FUNCTION_BLOCK "Sq_5.1"   // FB1511, GRAPH_PLUS
{ S7_Optimized_Access := 'TRUE' }
VERSION : 0.1
   VAR_INPUT
      OFF_SQ : Bool := false;   // Kette ausschalten
      INIT_SQ : Bool := false;   // Kette in Initialzustand versetzen
      ACK_EF : Bool := false;   // Alle Fehler und Störungen quittieren
      S_PREV : Bool := false;   // Vorherigen Schritt am Parameter S_NO ausgeben
      S_NEXT : Bool := false;   // Nächsten Schritt am Parameter S_NO anzeigen
      SW_AUTO : Bool := false;   // Automatischer Betrieb
      SW_TAP : Bool := false;   // Halbautomatisch/Weiterschalten mit Transition
      SW_TOP : Bool := false;   // Halbautomatisch/Ignoriere Transition
      SW_MAN : Bool := false;   // Handbetrieb
      S_SEL : Int := 0;   // Schritt auswählen, der an S_NO ausgegeben werden soll
      S_ON : Bool := false;   // Schritt aktivieren, der an Parameter S_NO anliegt
      S_OFF : Bool := false;   // Schritt deaktivieren, der an Parameter S_NO anliegt
      T_PUSH : Bool := false;   // Schaltfreigabe für Transition im halbautomatischen Betrieb
      itMaxRuntime : Time := t#10s;   // Maximale Laufzeit für diesen Prozess
   END_VAR
   VAR_OUTPUT
      S_NO : Int := 0;   // Schrittnummer
      S_MORE : Bool := false;   // Weitere Schritte sind vorhanden und können in S_NO angezeigt werden.
      S_ACTIVE : Bool := false;   // Schritt, der an Parameter S_NO angezeigt wird, ist aktiv
      ERR_FLT : Bool := false;   // Sammelfehler Interlock oder Supervision
      AUTO_ON : Bool := false;   // Automatischer Betrieb eingeschaltet
      TAP_ON : Bool := false;   // Halbautomatischer Betrieb/Schritt mit Transition eingeschaltet
      TOP_ON : Bool := false;   // Halbautomatischer Betrieb/Ignoriere Transition eingeschaltet
      MAN_ON : Bool := false;   // Handbetrieb eingeschaltet
      qxIsActive : Bool;   // Schrittkette läuft
      qxIsInHome : Bool;   // steht in Grundstellung
      qxConveyorIsEmpty : Bool;   // Linearförderer wurde geleert
      qxLackOfParts : Bool;   // Teilemangel
   END_VAR
   VAR_IN_OUT
      signals : "typeStationSignals";   // Stationssteuersignale
      sq : "typeStepSequence";   // Schrittkettensteuersignale
   END_VAR
   VAR
      sstReleaseCycle : Struct
         ErrorAck : Bool;
         No_LastCycle : Int;
         T : Time;   // Aktive Zeit des ReleaseCycle
         Tck : Time;
         TckPrev : Time;
      END_STRUCT;
      susiGripperState : USInt;
      sinstTofConveyorOn : TOF_TIME;
      sinstTonConveyorIsEmpty : TON_TIME;
      sinstTonPartInSep : TON_TIME;
      sinstTonLackOfParts : TON_TIME;
      sinstTonNoPartInSep : TON_TIME;
      sxConveyorOn : Bool;
      sxWaitForPart : Bool;
      HMI_INFO : Array[0..8] of UInt;
      IF_PAR : G7_IfParPlus_V6;
      RT_DATA : G7_RTDataPlus_V6;   // Interner Datenbereich
      Automatikablauf : G7_TransitionPlus_V6;   // Transitionsstruktur
      Freigabe : G7_TransitionPlus_V6;   // Transitionsstruktur
      GreiferLeer : G7_TransitionPlus_V6;   // Transitionsstruktur
      Fertig : G7_TransitionPlus_V6;   // Transitionsstruktur
      Grundstellungsfahrt : G7_TransitionPlus_V6;   // Transitionsstruktur
      GST_Aktiv : G7_TransitionPlus_V6;   // Transitionsstruktur
      GST_Beendet : G7_TransitionPlus_V6;   // Transitionsstruktur
      Beendet : G7_TransitionPlus_V6;   // Transitionsstruktur
      DoneToIndexer : G7_TransitionPlus_V6;   // Transitionsstruktur / Transition structure
      JogT1 : G7_TransitionPlus_V6;   // Transitionsstruktur / Transition structure
      JogT2 : G7_TransitionPlus_V6;   // Transitionsstruktur / Transition structure
      GS_CapsSourceStopperInHome : G7_TransitionPlus_V6;   // Transitionsstruktur / Transition structure
      GS_NotEmptying : G7_TransitionPlus_V6;   // Transitionsstruktur / Transition structure
      GS_Emptying : G7_TransitionPlus_V6;   // Transitionsstruktur / Transition structure
      GS_CapsSourceStopperInWork : G7_TransitionPlus_V6;   // Transitionsstruktur / Transition structure
      GS_AxisRInHome : G7_TransitionPlus_V6;   // Transitionsstruktur / Transition structure
      GS_AxisZ1InHome : G7_TransitionPlus_V6;   // Transitionsstruktur / Transition structure
      GS_AxisZ2InHome : G7_TransitionPlus_V6;   // Transitionsstruktur / Transition structure
      GS_AxisXInHome : G7_TransitionPlus_V6;   // Transitionsstruktur / Transition structure
      GS_GreiferUnbeladen : G7_TransitionPlus_V6;   // Transitionsstruktur / Transition structure
      GS_GreiferBeladen : G7_TransitionPlus_V6;   // Transitionsstruktur / Transition structure
      GS_GreiferUnbekannt : G7_TransitionPlus_V6;   // Transitionsstruktur / Transition structure
      GS_GripperInHome : G7_TransitionPlus_V6;   // Transitionsstruktur / Transition structure
      GS_GripperInWork : G7_TransitionPlus_V6;   // Transitionsstruktur / Transition structure
      GS_CapsSourceStopperInWork_1 : G7_TransitionPlus_V6;   // Transitionsstruktur / Transition structure
      GS_GripperInHome_1 : G7_TransitionPlus_V6;   // Transitionsstruktur / Transition structure
      CapsSourceStopperInHome_1 : G7_TransitionPlus_V6;   // Transitionsstruktur / Transition structure
      GS_GripperStatusIsEmpty : G7_TransitionPlus_V6;   // Transitionsstruktur / Transition structure
      NotEmptying : G7_TransitionPlus_V6;   // Transitionsstruktur / Transition structure
      Emptying : G7_TransitionPlus_V6;   // Transitionsstruktur / Transition structure
      CapsSourceStopperInWork_2 : G7_TransitionPlus_V6;   // Transitionsstruktur / Transition structure
      GripperInHome_2 : G7_TransitionPlus_V6;   // Transitionsstruktur / Transition structure
      GripperIsEmpty : G7_TransitionPlus_V6;   // Transitionsstruktur / Transition structure
      ConveyorIsEmpty : G7_TransitionPlus_V6;   // Transitionsstruktur / Transition structure
      SepEmpty : G7_TransitionPlus_V6;   // Transitionsstruktur / Transition structure
      SepNotEmpty : G7_TransitionPlus_V6;   // Transitionsstruktur / Transition structure
      CapsSourceStopperInHome : G7_TransitionPlus_V6;   // Transitionsstruktur / Transition structure
      AxisZ2InWork : G7_TransitionPlus_V6;   // Transitionsstruktur / Transition structure
      GripperInWork : G7_TransitionPlus_V6;   // Transitionsstruktur / Transition structure
      GripperIsLoaded : G7_TransitionPlus_V6;   // Transitionsstruktur / Transition structure
      AxisZ2InHome : G7_TransitionPlus_V6;   // Transitionsstruktur / Transition structure
      JogT3 : G7_TransitionPlus_V6;   // Transitionsstruktur / Transition structure
      JogT4 : G7_TransitionPlus_V6;   // Transitionsstruktur / Transition structure
      JogT5 : G7_TransitionPlus_V6;   // Transitionsstruktur / Transition structure
      SeparatorIsEmpty : G7_TransitionPlus_V6;   // Transitionsstruktur / Transition structure
      ConvEmptyIsSet : G7_TransitionPlus_V6;   // Transitionsstruktur / Transition structure
      JogT6 : G7_TransitionPlus_V6;   // Transitionsstruktur / Transition structure
      GripperIsLoaded_1 : G7_TransitionPlus_V6;   // Transitionsstruktur / Transition structure
      GripperIsEmpty_1 : G7_TransitionPlus_V6;   // Transitionsstruktur / Transition structure
      CapsSourceStopperInHome_2 : G7_TransitionPlus_V6;   // Transitionsstruktur / Transition structure
      GripperInWork_1 : G7_TransitionPlus_V6;   // Transitionsstruktur / Transition structure
      GripperIsLoaded_2 : G7_TransitionPlus_V6;   // Transitionsstruktur / Transition structure
      PartInSeparator_2 : G7_TransitionPlus_V6;   // Transitionsstruktur / Transition structure
      AxisZ2InWork_2 : G7_TransitionPlus_V6;   // Transitionsstruktur / Transition structure
      AxisZ2InHome_1 : G7_TransitionPlus_V6;   // Transitionsstruktur / Transition structure
      SeparatorIsEmpty_1 : G7_TransitionPlus_V6;   // Transitionsstruktur / Transition structure
      JogT7 : G7_TransitionPlus_V6;   // Transitionsstruktur / Transition structure
      JogT8 : G7_TransitionPlus_V6;   // Transitionsstruktur / Transition structure
      JogT9 : G7_TransitionPlus_V6;   // Transitionsstruktur / Transition structure
      AxisXInWork : G7_TransitionPlus_V6;   // Transitionsstruktur / Transition structure
      AxisRInWork : G7_TransitionPlus_V6;   // Transitionsstruktur / Transition structure
      AxisZ1InWork : G7_TransitionPlus_V6;   // Transitionsstruktur / Transition structure
      GripperInHome_3 : G7_TransitionPlus_V6;   // Transitionsstruktur / Transition structure
      GripperIsEmpty_2 : G7_TransitionPlus_V6;   // Transitionsstruktur / Transition structure
      AxisZ1InHome : G7_TransitionPlus_V6;   // Transitionsstruktur / Transition structure
      GS_AxisRInHome_1 : G7_TransitionPlus_V6;   // Transitionsstruktur / Transition structure
      AxisXInHome : G7_TransitionPlus_V6;   // Transitionsstruktur / Transition structure
      JogT10 : G7_TransitionPlus_V6;   // Transitionsstruktur / Transition structure
      JogT11 : G7_TransitionPlus_V6;   // Transitionsstruktur / Transition structure
      JogT12 : G7_TransitionPlus_V6;   // Transitionsstruktur / Transition structure
      JogT13 : G7_TransitionPlus_V6;   // Transitionsstruktur / Transition structure
      JogT14 : G7_TransitionPlus_V6;   // Transitionsstruktur / Transition structure
      JogT15 : G7_TransitionPlus_V6;   // Transitionsstruktur / Transition structure
      Initialschritt : G7_StepPlus_V6;   // Schrittstruktur
      Grundstellung : G7_StepPlus_V6;   // Schrittstruktur
      SK_läuft : G7_StepPlus_V6;   // Schrittstruktur
      Fertigmeldung : G7_StepPlus_V6;   // Schrittstruktur
      "Start Grundstellungsfahrt" : G7_StepPlus_V6;   // Schrittstruktur
      "Fertig Grundstellungsfahrt" : G7_StepPlus_V6;   // Schrittstruktur
      Ende : G7_StepPlus_V6;   // Schrittstruktur
      ResetRelease : G7_StepPlus_V6;   // Schrittstruktur / Step structure
      JogS1 : G7_StepPlus_V6;   // Schrittstruktur / Step structure
      JogS2 : G7_StepPlus_V6;   // Schrittstruktur / Step structure
      GS_CapsSourceStopperHomePos : G7_StepPlus_V6;   // Schrittstruktur / Step structure
      "GS_Emptying?" : G7_StepPlus_V6;   // Schrittstruktur / Step structure
      GS_CapsSourceStopperWorkPos : G7_StepPlus_V6;   // Schrittstruktur / Step structure
      GS_AxisRHomePos : G7_StepPlus_V6;   // Schrittstruktur / Step structure
      GS_AxisZ1HomePos : G7_StepPlus_V6;   // Schrittstruktur / Step structure
      GS_AxisZ2HomePos : G7_StepPlus_V6;   // Schrittstruktur / Step structure
      GS_AxisXHomePos : G7_StepPlus_V6;   // Schrittstruktur / Step structure
      GS_GripperState : G7_StepPlus_V6;   // Schrittstruktur / Step structure
      GS_GripperHomePos : G7_StepPlus_V6;   // Schrittstruktur / Step structure
      GS_GripperWorkPos : G7_StepPlus_V6;   // Schrittstruktur / Step structure
      GS_CapsSourceStopperWorkPos_1 : G7_StepPlus_V6;   // Schrittstruktur / Step structure
      GS_GripperHomePos_1 : G7_StepPlus_V6;   // Schrittstruktur / Step structure
      GS_CapsSourceStopperHomePos_1 : G7_StepPlus_V6;   // Schrittstruktur / Step structure
      GS_GripperStatusEmpty : G7_StepPlus_V6;   // Schrittstruktur / Step structure
      "Emptying?" : G7_StepPlus_V6;   // Schrittstruktur / Step structure
      CapsSourceStopperWorkPos : G7_StepPlus_V6;   // Schrittstruktur / Step structure
      GripperHomePos : G7_StepPlus_V6;   // Schrittstruktur / Step structure
      GripperEmpty : G7_StepPlus_V6;   // Schrittstruktur / Step structure
      EmptyingConveyor : G7_StepPlus_V6;   // Schrittstruktur / Step structure
      SeparatorEmpty : G7_StepPlus_V6;   // Schrittstruktur / Step structure
      CapsSourceStopperHomePos : G7_StepPlus_V6;   // Schrittstruktur / Step structure
      AxisZ2WorkPos : G7_StepPlus_V6;   // Schrittstruktur / Step structure
      GripperWorkPos : G7_StepPlus_V6;   // Schrittstruktur / Step structure
      GripperLoaded : G7_StepPlus_V6;   // Schrittstruktur / Step structure
      AxisZ2HomePos : G7_StepPlus_V6;   // Schrittstruktur / Step structure
      JogS3 : G7_StepPlus_V6;   // Schrittstruktur / Step structure
      JogS4 : G7_StepPlus_V6;   // Schrittstruktur / Step structure
      JogS5 : G7_StepPlus_V6;   // Schrittstruktur / Step structure
      CheckSepEmpty : G7_StepPlus_V6;   // Schrittstruktur / Step structure
      SetConvEmpty : G7_StepPlus_V6;   // Schrittstruktur / Step structure
      JogS6 : G7_StepPlus_V6;   // Schrittstruktur / Step structure
      GripperState : G7_StepPlus_V6;   // Schrittstruktur / Step structure
      CapsSourceStopperHomePos_1 : G7_StepPlus_V6;   // Schrittstruktur / Step structure
      GripperWorkPos_1 : G7_StepPlus_V6;   // Schrittstruktur / Step structure
      GripperLoaded_1 : G7_StepPlus_V6;   // Schrittstruktur / Step structure
      SeparatorBusy_1 : G7_StepPlus_V6;   // Schrittstruktur / Step structure
      AxisZ2WorkPos_2 : G7_StepPlus_V6;   // Schrittstruktur / Step structure
      AxisZ2HomePos_1 : G7_StepPlus_V6;   // Schrittstruktur / Step structure
      CheckSepEmpty_1 : G7_StepPlus_V6;   // Schrittstruktur / Step structure
      JogS7 : G7_StepPlus_V6;   // Schrittstruktur / Step structure
      JogS8 : G7_StepPlus_V6;   // Schrittstruktur / Step structure
      JogS9 : G7_StepPlus_V6;   // Schrittstruktur / Step structure
      AxisXWorkPos : G7_StepPlus_V6;   // Schrittstruktur / Step structure
      AxisRWorkPos : G7_StepPlus_V6;   // Schrittstruktur / Step structure
      AxisZ1WorkPos : G7_StepPlus_V6;   // Schrittstruktur / Step structure
      GripperHomePos_1 : G7_StepPlus_V6;   // Schrittstruktur / Step structure
      GripperEmpty_1 : G7_StepPlus_V6;   // Schrittstruktur / Step structure
      AxisZ1HomePos : G7_StepPlus_V6;   // Schrittstruktur / Step structure
      GS_AxisRHomePos_1 : G7_StepPlus_V6;   // Schrittstruktur / Step structure
      AxisXHomePos : G7_StepPlus_V6;   // Schrittstruktur / Step structure
      JogS10 : G7_StepPlus_V6;   // Schrittstruktur / Step structure
      JogS11 : G7_StepPlus_V6;   // Schrittstruktur / Step structure
      JogS12 : G7_StepPlus_V6;   // Schrittstruktur / Step structure
      JogS13 : G7_StepPlus_V6;   // Schrittstruktur / Step structure
      JogS14 : G7_StepPlus_V6;   // Schrittstruktur / Step structure
      JogS15 : G7_StepPlus_V6;   // Schrittstruktur / Step structure
      SINI : Array[0..1] of USInt;
      LSTT : Array[0..72] of USInt;
      ATAJ : Array[0..72] of USInt;
      ATAB : Array[0..72] of USInt;
      PSTT : Array[0..72] of USInt;
      NSTT : Array[0..72] of USInt;
      ASSJ : Array[0..65] of USInt;
      ASSB : Array[0..65] of USInt;
      PTTS : Array[0..65] of USInt;
      NTTS : Array[0..65] of USInt;
      SW_SQTS : Array[0..65] of USInt;
      SWITCH : Array[0..40] of USInt;
      TVX : Array[0..14] of USInt;
      TTX : Array[0..14] of USInt;
      TSX : Array[0..1] of USInt;
      S00X : Array[0..1] of USInt;
      SOFFX : Array[0..1] of USInt;
      SONX : Array[0..1] of USInt;
      SAX : Array[0..1] of USInt;
      SERRX : Array[0..66] of USInt;
      SMX : Array[0..66] of USInt;
      S0X : Array[0..66] of USInt;
      S1X : Array[0..66] of USInt;
      IL_ALARM_INST : Diag_Alarm;
      SUP_ALARM_INST : Diag_Alarm;
      STEP_TIME_ALARM_INST : Diag_Alarm;
      IEC_TIMER_INST : IEC_TIMER;
      TRANSACTION_FLAG : Bool := false;
   END_VAR
   VAR_TEMP
      txStartCondition : Bool;
      tdTckDiff : DInt;
   END_VAR
   VAR CONSTANT
      GRIPPER_UNKNOWN : USInt := 0;   // Greiferstatus "unbekannt"
      GRIPPER_EMPTY : USInt := 1;   // Greiferstatus "leer"
      GRIPPER_LOADED : USInt := 2;   // Greiferstatus "beladen"
   END_VAR
   VAR_TEMP   // added for the SCL form of the ladder/FBD networks
      _w1 : Bool;
      _w2 : Bool;
   END_VAR
   // SINI[0] := 2;
   // LSTT[0] := 255;
   // LSTT[1] := 255;
   // LSTT[2] := 255;
   // LSTT[3] := 255;
   // LSTT[4] := 255;
   // LSTT[5] := 255;
   // LSTT[6] := 255;
   // LSTT[7] := 1;
   // ATAJ[1] := 1;
   // ATAJ[2] := 2;
   // ATAJ[3] := 6;
   // ATAJ[4] := 4;
   // ATAJ[5] := 5;
   // ATAJ[6] := 3;
   // ATAJ[7] := 7;
   // ATAB[0] := 4;
   // ATAB[1] := 1;
   // ATAB[2] := 2;
   // ATAB[3] := 3;
   // ATAB[5] := 5;
   // ATAB[6] := 6;
   // ATAB[7] := 7;
   // PSTT[1] := 1;
   // PSTT[2] := 2;
   // PSTT[3] := 3;
   // PSTT[5] := 4;
   // PSTT[6] := 5;
   // PSTT[7] := 6;
   // NSTT[0] := 1;
   // NSTT[1] := 2;
   // NSTT[2] := 24;
   // NSTT[3] := 6;
   // NSTT[4] := 4;
   // NSTT[5] := 14;
   // NSTT[6] := 6;
   // NSTT[7] := 1;
   // ASSJ[1] := 1;
   // ASSJ[2] := 2;
   // ASSJ[3] := 3;
   // ASSJ[4] := 4;
   // ASSJ[5] := 5;
   // ASSJ[6] := 6;
   // ASSB[1] := 1;
   // ASSB[2] := 2;
   // ASSB[3] := 3;
   // ASSB[4] := 4;
   // ASSB[5] := 5;
   // ASSB[6] := 6;
   // PTTS[0] := 255;
   // PTTS[2] := 1;
   // PTTS[3] := 8;
   // PTTS[4] := 4;
   // PTTS[5] := 11;
   // PTTS[6] := 3;
   // NTTS[1] := 1;
   // NTTS[2] := 2;
   // NTTS[3] := 3;
   // NTTS[4] := 5;
   // NTTS[5] := 6;
   // NTTS[6] := 7;
   // SW_SQTS[1] := 1;
   // SW_SQTS[2] := 1;
   // SW_SQTS[3] := 2;
   // SW_SQTS[4] := 3;
   // SW_SQTS[5] := 4;
   // SW_SQTS[6] := 5;
   // TVX[0] := 16#1;
   // TTX[0] := 16#1;
   // TSX[0] := 16#1;
   // S00X[0] := 16#1;
   // SOFFX[0] := 16#1;
   // SONX[0] := 16#1;
   // SAX[0] := 16#1;
   // SERRX[0] := 16#1;
   // SMX[0] := 16#1;
   // S0X[0] := 16#1;
   // S1X[0] := 16#1;
   // LSTT[8] := 255;
   // ATAJ[8] := 58;
   // ATAB[8] := 8;
   // PSTT[8] := 7;
   // NSTT[8] := 3;
   // ASSJ[7] := 7;
   // ASSB[7] := 7;
   // PTTS[7] := 66;
   // NTTS[7] := 8;
   // SW_SQTS[7] := 6;
   // LSTT[9] := 255;
   // ATAJ[9] := 9;
   // ATAB[9] := 9;
   // PSTT[9] := 8;
   // NSTT[9] := 26;
   // ASSJ[8] := 8;
   // ASSB[8] := 8;
   // PTTS[8] := 30;
   // NTTS[8] := 9;
   // SW_SQTS[8] := 7;
   // LSTT[10] := 255;
   // LSTT[11] := 255;
   // LSTT[12] := 255;
   // ATAJ[10] := 10;
   // ATAJ[11] := 14;
   // ATAJ[12] := 12;
   // ATAB[10] := 10;
   // ATAB[11] := 11;
   // ATAB[12] := 13;
   // PSTT[10] := 9;
   // PSTT[11] := 10;
   // PSTT[12] := 11;
   // NSTT[10] := 28;
   // NSTT[11] := 5;
   // NSTT[12] := 10;
   // ASSJ[9] := 9;
   // ASSJ[10] := 10;
   // ASSJ[11] := 11;
   // ASSB[9] := 9;
   // ASSB[10] := 10;
   // ASSB[11] := 11;
   // PTTS[9] := 32;
   // PTTS[10] := 12;
   // PTTS[11] := 22;
   // NTTS[9] := 10;
   // NTTS[10] := 11;
   // NTTS[11] := 12;
   // SW_SQTS[9] := 7;
   // SW_SQTS[10] := 8;
   // SW_SQTS[11] := 9;
   // LSTT[13] := 255;
   // ATAJ[13] := 13;
   // ATAB[13] := 12;
   // PSTT[13] := 11;
   // NSTT[13] := 12;
   // ASSJ[12] := 12;
   // ASSB[12] := 12;
   // PTTS[12] := 13;
   // NTTS[12] := 14;
   // SW_SQTS[12] := 10;
   // LSTT[14] := 255;
   // LSTT[15] := 255;
   // LSTT[16] := 255;
   // LSTT[17] := 255;
   // LSTT[18] := 255;
   // LSTT[19] := 255;
   // LSTT[20] := 255;
   // LSTT[21] := 255;
   // LSTT[22] := 255;
   // LSTT[23] := 255;
   // LSTT[24] := 255;
   // LSTT[25] := 255;
   // LSTT[26] := 255;
   // LSTT[27] := 255;
   // ATAJ[14] := 11;
   // ATAJ[15] := 15;
   // ATAJ[16] := 16;
   // ATAJ[17] := 17;
   // ATAJ[18] := 18;
   // ATAJ[19] := 19;
   // ATAJ[20] := 20;
   // ATAJ[21] := 21;
   // ATAJ[22] := 23;
   // ATAJ[23] := 26;
   // ATAJ[24] := 24;
   // ATAJ[25] := 25;
   // ATAJ[26] := 22;
   // ATAJ[27] := 27;
   // ATAB[14] := 14;
   // ATAB[15] := 15;
   // ATAB[16] := 16;
   // ATAB[17] := 17;
   // ATAB[18] := 18;
   // ATAB[19] := 20;
   // ATAB[20] := 21;
   // ATAB[21] := 19;
   // ATAB[22] := 22;
   // ATAB[23] := 23;
   // ATAB[24] := 24;
   // ATAB[25] := 25;
   // ATAB[26] := 26;
   // ATAB[27] := 27;
   // PSTT[14] := 12;
   // PSTT[15] := 13;
   // PSTT[16] := 14;
   // PSTT[17] := 15;
   // PSTT[18] := 16;
   // PSTT[19] := 17;
   // PSTT[20] := 17;
   // PSTT[21] := 17;
   // PSTT[22] := 18;
   // PSTT[23] := 19;
   // PSTT[24] := 20;
   // PSTT[25] := 21;
   // PSTT[26] := 22;
   // PSTT[27] := 23;
   // NSTT[14] := 5;
   // NSTT[15] := 17;
   // NSTT[16] := 15;
   // NSTT[17] := 16;
   // NSTT[18] := 13;
   // NSTT[19] := 18;
   // NSTT[20] := 19;
   // NSTT[21] := 20;
   // NSTT[22] := 11;
   // NSTT[23] := 11;
   // NSTT[24] := 21;
   // NSTT[25] := 23;
   // NSTT[26] := 11;
   // NSTT[27] := 22;
   // ASSJ[13] := 13;
   // ASSJ[14] := 14;
   // ASSJ[15] := 15;
   // ASSJ[16] := 16;
   // ASSJ[17] := 17;
   // ASSJ[18] := 18;
   // ASSJ[19] := 19;
   // ASSJ[20] := 20;
   // ASSJ[21] := 21;
   // ASSJ[22] := 22;
   // ASSJ[23] := 23;
   // ASSB[13] := 13;
   // ASSB[14] := 14;
   // ASSB[15] := 15;
   // ASSB[16] := 16;
   // ASSB[17] := 17;
   // ASSB[18] := 18;
   // ASSB[19] := 19;
   // ASSB[20] := 20;
   // ASSB[21] := 21;
   // ASSB[22] := 22;
   // ASSB[23] := 23;
   // PTTS[13] := 18;
   // PTTS[14] := 5;
   // PTTS[15] := 16;
   // PTTS[16] := 17;
   // PTTS[17] := 15;
   // PTTS[18] := 19;
   // PTTS[19] := 20;
   // PTTS[20] := 21;
   // PTTS[21] := 24;
   // PTTS[22] := 27;
   // PTTS[23] := 25;
   // NTTS[13] := 15;
   // NTTS[14] := 16;
   // NTTS[15] := 17;
   // NTTS[16] := 18;
   // NTTS[17] := 19;
   // NTTS[18] := 22;
   // NTTS[19] := 23;
   // NTTS[20] := 24;
   // NTTS[21] := 25;
   // NTTS[22] := 26;
   // NTTS[23] := 27;
   // SW_SQTS[13] := 3;
   // SW_SQTS[14] := 3;
   // SW_SQTS[15] := 3;
   // SW_SQTS[16] := 3;
   // SW_SQTS[17] := 3;
   // SW_SQTS[18] := 11;
   // SW_SQTS[19] := 12;
   // SW_SQTS[20] := 13;
   // SW_SQTS[21] := 13;
   // SW_SQTS[22] := 13;
   // SW_SQTS[23] := 13;
   // LSTT[28] := 255;
   // LSTT[29] := 255;
   // LSTT[30] := 255;
   // LSTT[31] := 255;
   // LSTT[32] := 255;
   // LSTT[33] := 255;
   // LSTT[34] := 255;
   // LSTT[35] := 255;
   // LSTT[36] := 255;
   // LSTT[37] := 255;
   // LSTT[38] := 255;
   // LSTT[39] := 255;
   // LSTT[40] := 255;
   // LSTT[41] := 255;
   // LSTT[42] := 255;
   // LSTT[43] := 255;
   // ATAJ[28] := 28;
   // ATAJ[29] := 29;
   // ATAJ[30] := 30;
   // ATAJ[31] := 31;
   // ATAJ[32] := 32;
   // ATAJ[33] := 33;
   // ATAJ[34] := 34;
   // ATAJ[35] := 35;
   // ATAJ[36] := 36;
   // ATAJ[37] := 37;
   // ATAJ[38] := 38;
   // ATAJ[39] := 39;
   // ATAJ[40] := 40;
   // ATAJ[41] := 41;
   // ATAJ[42] := 42;
   // ATAJ[43] := 43;
   // ATAB[28] := 29;
   // ATAB[29] := 28;
   // ATAB[30] := 30;
   // ATAB[31] := 31;
   // ATAB[32] := 32;
   // ATAB[33] := 33;
   // ATAB[34] := 35;
   // ATAB[35] := 34;
   // ATAB[36] := 36;
   // ATAB[37] := 37;
   // ATAB[38] := 38;
   // ATAB[39] := 39;
   // ATAB[40] := 40;
   // ATAB[41] := 41;
   // ATAB[42] := 42;
   // ATAB[43] := 43;
   // PSTT[28] := 24;
   // PSTT[29] := 24;
   // PSTT[30] := 25;
   // PSTT[31] := 26;
   // PSTT[32] := 27;
   // PSTT[33] := 28;
   // PSTT[34] := 29;
   // PSTT[35] := 29;
   // PSTT[36] := 30;
   // PSTT[37] := 31;
   // PSTT[38] := 32;
   // PSTT[39] := 33;
   // PSTT[40] := 34;
   // PSTT[41] := 35;
   // PSTT[42] := 36;
   // PSTT[43] := 37;
   // NSTT[28] := 42;
   // NSTT[29] := 29;
   // NSTT[30] := 8;
   // NSTT[31] := 27;
   // NSTT[32] := 9;
   // NSTT[33] := 39;
   // NSTT[34] := 25;
   // NSTT[35] := 30;
   // NSTT[36] := 35;
   // NSTT[37] := 36;
   // NSTT[38] := 33;
   // NSTT[39] := 37;
   // NSTT[40] := 38;
   // NSTT[41] := 31;
   // NSTT[42] := 32;
   // NSTT[43] := 34;
   // ASSJ[24] := 24;
   // ASSJ[25] := 25;
   // ASSJ[26] := 26;
   // ASSJ[27] := 27;
   // ASSJ[28] := 28;
   // ASSJ[29] := 29;
   // ASSJ[30] := 30;
   // ASSJ[31] := 31;
   // ASSJ[32] := 32;
   // ASSJ[33] := 33;
   // ASSJ[34] := 34;
   // ASSJ[35] := 35;
   // ASSJ[36] := 36;
   // ASSJ[37] := 37;
   // ASSB[24] := 24;
   // ASSB[25] := 25;
   // ASSB[26] := 26;
   // ASSB[27] := 27;
   // ASSB[28] := 28;
   // ASSB[29] := 29;
   // ASSB[30] := 30;
   // ASSB[31] := 31;
   // ASSB[32] := 32;
   // ASSB[33] := 33;
   // ASSB[34] := 34;
   // ASSB[35] := 35;
   // ASSB[36] := 36;
   // ASSB[37] := 37;
   // PTTS[24] := 2;
   // PTTS[25] := 34;
   // PTTS[26] := 9;
   // PTTS[27] := 31;
   // PTTS[28] := 10;
   // PTTS[29] := 29;
   // PTTS[30] := 35;
   // PTTS[31] := 41;
   // PTTS[32] := 42;
   // PTTS[33] := 38;
   // PTTS[34] := 43;
   // PTTS[35] := 36;
   // PTTS[36] := 37;
   // PTTS[37] := 39;
   // NTTS[24] := 28;
   // NTTS[25] := 30;
   // NTTS[26] := 31;
   // NTTS[27] := 32;
   // NTTS[28] := 33;
   // NTTS[29] := 34;
   // NTTS[30] := 36;
   // NTTS[31] := 37;
   // NTTS[32] := 38;
   // NTTS[33] := 39;
   // NTTS[34] := 40;
   // NTTS[35] := 41;
   // NTTS[36] := 42;
   // NTTS[37] := 43;
   // SW_SQTS[24] := 1;
   // SW_SQTS[25] := 7;
   // SW_SQTS[26] := 7;
   // SW_SQTS[27] := 7;
   // SW_SQTS[28] := 7;
   // SW_SQTS[29] := 14;
   // SW_SQTS[30] := 15;
   // SW_SQTS[31] := 15;
   // SW_SQTS[32] := 15;
   // SW_SQTS[33] := 15;
   // SW_SQTS[34] := 15;
   // SW_SQTS[35] := 15;
   // SW_SQTS[36] := 15;
   // SW_SQTS[37] := 15;
   // LSTT[44] := 255;
   // LSTT[45] := 255;
   // LSTT[46] := 29;
   // LSTT[47] := 255;
   // LSTT[48] := 255;
   // LSTT[49] := 255;
   // LSTT[50] := 255;
   // LSTT[51] := 255;
   // LSTT[52] := 255;
   // LSTT[53] := 255;
   // LSTT[54] := 255;
   // LSTT[55] := 255;
   // LSTT[56] := 255;
   // LSTT[57] := 255;
   // LSTT[58] := 255;
   // LSTT[59] := 255;
   // LSTT[60] := 255;
   // LSTT[61] := 255;
   // LSTT[62] := 255;
   // LSTT[63] := 255;
   // LSTT[64] := 255;
   // LSTT[65] := 255;
   // LSTT[66] := 255;
   // LSTT[67] := 255;
   // LSTT[68] := 255;
   // LSTT[69] := 255;
   // LSTT[70] := 255;
   // LSTT[71] := 255;
   // LSTT[72] := 255;
   // ATAJ[44] := 44;
   // ATAJ[45] := 8;
   // ATAJ[46] := 46;
   // ATAJ[47] := 47;
   // ATAJ[48] := 48;
   // ATAJ[49] := 49;
   // ATAJ[50] := 50;
   // ATAJ[51] := 51;
   // ATAJ[52] := 52;
   // ATAJ[53] := 53;
   // ATAJ[54] := 54;
   // ATAJ[55] := 55;
   // ATAJ[56] := 56;
   // ATAJ[57] := 57;
   // ATAJ[58] := 45;
   // ATAJ[59] := 59;
   // ATAJ[60] := 60;
   // ATAJ[61] := 61;
   // ATAJ[62] := 62;
   // ATAJ[63] := 63;
   // ATAJ[64] := 64;
   // ATAJ[65] := 65;
   // ATAJ[66] := 66;
   // ATAJ[67] := 67;
   // ATAJ[68] := 68;
   // ATAJ[69] := 69;
   // ATAJ[70] := 70;
   // ATAJ[71] := 71;
   // ATAJ[72] := 72;
   // ATAB[44] := 44;
   // ATAB[45] := 45;
   // ATAB[46] := 46;
   // ATAB[47] := 48;
   // ATAB[48] := 47;
   // ATAB[49] := 49;
   // ATAB[50] := 50;
   // ATAB[51] := 51;
   // ATAB[52] := 52;
   // ATAB[53] := 53;
   // ATAB[54] := 54;
   // ATAB[55] := 55;
   // ATAB[56] := 56;
   // ATAB[57] := 57;
   // ATAB[58] := 58;
   // ATAB[59] := 59;
   // ATAB[60] := 60;
   // ATAB[61] := 61;
   // ATAB[62] := 62;
   // ATAB[63] := 63;
   // ATAB[64] := 64;
   // ATAB[65] := 65;
   // ATAB[66] := 66;
   // ATAB[67] := 67;
   // ATAB[68] := 68;
   // ATAB[69] := 69;
   // ATAB[70] := 70;
   // ATAB[71] := 71;
   // ATAB[72] := 72;
   // PSTT[44] := 38;
   // PSTT[45] := 39;
   // PSTT[46] := 40;
   // PSTT[47] := 41;
   // PSTT[48] := 41;
   // PSTT[49] := 42;
   // PSTT[50] := 43;
   // PSTT[51] := 44;
   // PSTT[52] := 45;
   // PSTT[53] := 46;
   // PSTT[54] := 47;
   // PSTT[55] := 48;
   // PSTT[56] := 49;
   // PSTT[57] := 50;
   // PSTT[58] := 51;
   // PSTT[59] := 52;
   // PSTT[60] := 53;
   // PSTT[61] := 54;
   // PSTT[62] := 55;
   // PSTT[63] := 56;
   // PSTT[64] := 57;
   // PSTT[65] := 58;
   // PSTT[66] := 59;
   // PSTT[67] := 60;
   // PSTT[68] := 61;
   // PSTT[69] := 62;
   // PSTT[70] := 63;
   // PSTT[71] := 64;
   // PSTT[72] := 65;
   // NSTT[44] := 40;
   // NSTT[45] := 3;
   // NSTT[46] := 29;
   // NSTT[47] := 52;
   // NSTT[48] := 45;
   // NSTT[49] := 41;
   // NSTT[50] := 44;
   // NSTT[51] := 50;
   // NSTT[52] := 46;
   // NSTT[53] := 49;
   // NSTT[54] := 48;
   // NSTT[55] := 51;
   // NSTT[56] := 43;
   // NSTT[57] := 47;
   // NSTT[58] := 3;
   // NSTT[59] := 60;
   // NSTT[60] := 61;
   // NSTT[61] := 62;
   // NSTT[62] := 56;
   // NSTT[63] := 63;
   // NSTT[64] := 64;
   // NSTT[65] := 65;
   // NSTT[66] := 7;
   // NSTT[67] := 53;
   // NSTT[68] := 54;
   // NSTT[69] := 55;
   // NSTT[70] := 57;
   // NSTT[71] := 58;
   // NSTT[72] := 59;
   // ASSJ[38] := 38;
   // ASSJ[39] := 39;
   // ASSJ[40] := 40;
   // ASSJ[41] := 41;
   // ASSJ[42] := 42;
   // ASSJ[43] := 43;
   // ASSJ[44] := 44;
   // ASSJ[45] := 45;
   // ASSJ[46] := 46;
   // ASSJ[47] := 47;
   // ASSJ[48] := 48;
   // ASSJ[49] := 49;
   // ASSJ[50] := 50;
   // ASSJ[51] := 51;
   // ASSJ[52] := 52;
   // ASSJ[53] := 53;
   // ASSJ[54] := 54;
   // ASSJ[55] := 55;
   // ASSJ[56] := 56;
   // ASSJ[57] := 57;
   // ASSJ[58] := 58;
   // ASSJ[59] := 59;
   // ASSJ[60] := 60;
   // ASSJ[61] := 61;
   // ASSJ[62] := 62;
   // ASSJ[63] := 63;
   // ASSJ[64] := 64;
   // ASSJ[65] := 65;
   // ASSB[38] := 38;
   // ASSB[39] := 39;
   // ASSB[40] := 40;
   // ASSB[41] := 41;
   // ASSB[42] := 42;
   // ASSB[43] := 43;
   // ASSB[44] := 44;
   // ASSB[45] := 45;
   // ASSB[46] := 46;
   // ASSB[47] := 47;
   // ASSB[48] := 48;
   // ASSB[49] := 49;
   // ASSB[50] := 50;
   // ASSB[51] := 51;
   // ASSB[52] := 52;
   // ASSB[53] := 53;
   // ASSB[54] := 54;
   // ASSB[55] := 55;
   // ASSB[56] := 56;
   // ASSB[57] := 57;
   // ASSB[58] := 58;
   // ASSB[59] := 59;
   // ASSB[60] := 60;
   // ASSB[61] := 61;
   // ASSB[62] := 62;
   // ASSB[63] := 63;
   // ASSB[64] := 64;
   // ASSB[65] := 65;
   // PTTS[38] := 40;
   // PTTS[39] := 33;
   // PTTS[40] := 44;
   // PTTS[41] := 49;
   // PTTS[42] := 28;
   // PTTS[43] := 56;
   // PTTS[44] := 50;
   // PTTS[45] := 48;
   // PTTS[46] := 52;
   // PTTS[47] := 57;
   // PTTS[48] := 54;
   // PTTS[49] := 53;
   // PTTS[50] := 51;
   // PTTS[51] := 55;
   // PTTS[52] := 47;
   // PTTS[53] := 67;
   // PTTS[54] := 68;
   // PTTS[55] := 69;
   // PTTS[56] := 62;
   // PTTS[57] := 70;
   // PTTS[58] := 71;
   // PTTS[59] := 72;
   // PTTS[60] := 59;
   // PTTS[61] := 60;
   // PTTS[62] := 61;
   // PTTS[63] := 63;
   // PTTS[64] := 64;
   // PTTS[65] := 65;
   // NTTS[38] := 44;
   // NTTS[39] := 45;
   // NTTS[40] := 46;
   // NTTS[41] := 47;
   // NTTS[42] := 49;
   // NTTS[43] := 50;
   // NTTS[44] := 51;
   // NTTS[45] := 52;
   // NTTS[46] := 53;
   // NTTS[47] := 54;
   // NTTS[48] := 55;
   // NTTS[49] := 56;
   // NTTS[50] := 57;
   // NTTS[51] := 58;
   // NTTS[52] := 59;
   // NTTS[53] := 60;
   // NTTS[54] := 61;
   // NTTS[55] := 62;
   // NTTS[56] := 63;
   // NTTS[57] := 64;
   // NTTS[58] := 65;
   // NTTS[59] := 66;
   // NTTS[60] := 67;
   // NTTS[61] := 68;
   // NTTS[62] := 69;
   // NTTS[63] := 70;
   // NTTS[64] := 71;
   // NTTS[65] := 72;
   // SW_SQTS[38] := 15;
   // SW_SQTS[39] := 7;
   // SW_SQTS[40] := 15;
   // SW_SQTS[41] := 16;
   // SW_SQTS[42] := 16;
   // SW_SQTS[43] := 17;
   // SW_SQTS[44] := 17;
   // SW_SQTS[45] := 17;
   // SW_SQTS[46] := 17;
   // SW_SQTS[47] := 17;
   // SW_SQTS[48] := 17;
   // SW_SQTS[49] := 17;
   // SW_SQTS[50] := 17;
   // SW_SQTS[51] := 17;
   // SW_SQTS[52] := 6;
   // SW_SQTS[53] := 6;
   // SW_SQTS[54] := 6;
   // SW_SQTS[55] := 6;
   // SW_SQTS[56] := 6;
   // SW_SQTS[57] := 6;
   // SW_SQTS[58] := 6;
   // SW_SQTS[59] := 6;
   // SW_SQTS[60] := 6;
   // SW_SQTS[61] := 6;
   // SW_SQTS[62] := 6;
   // SW_SQTS[63] := 6;
   // SW_SQTS[64] := 6;
   // SW_SQTS[65] := 6;
BEGIN
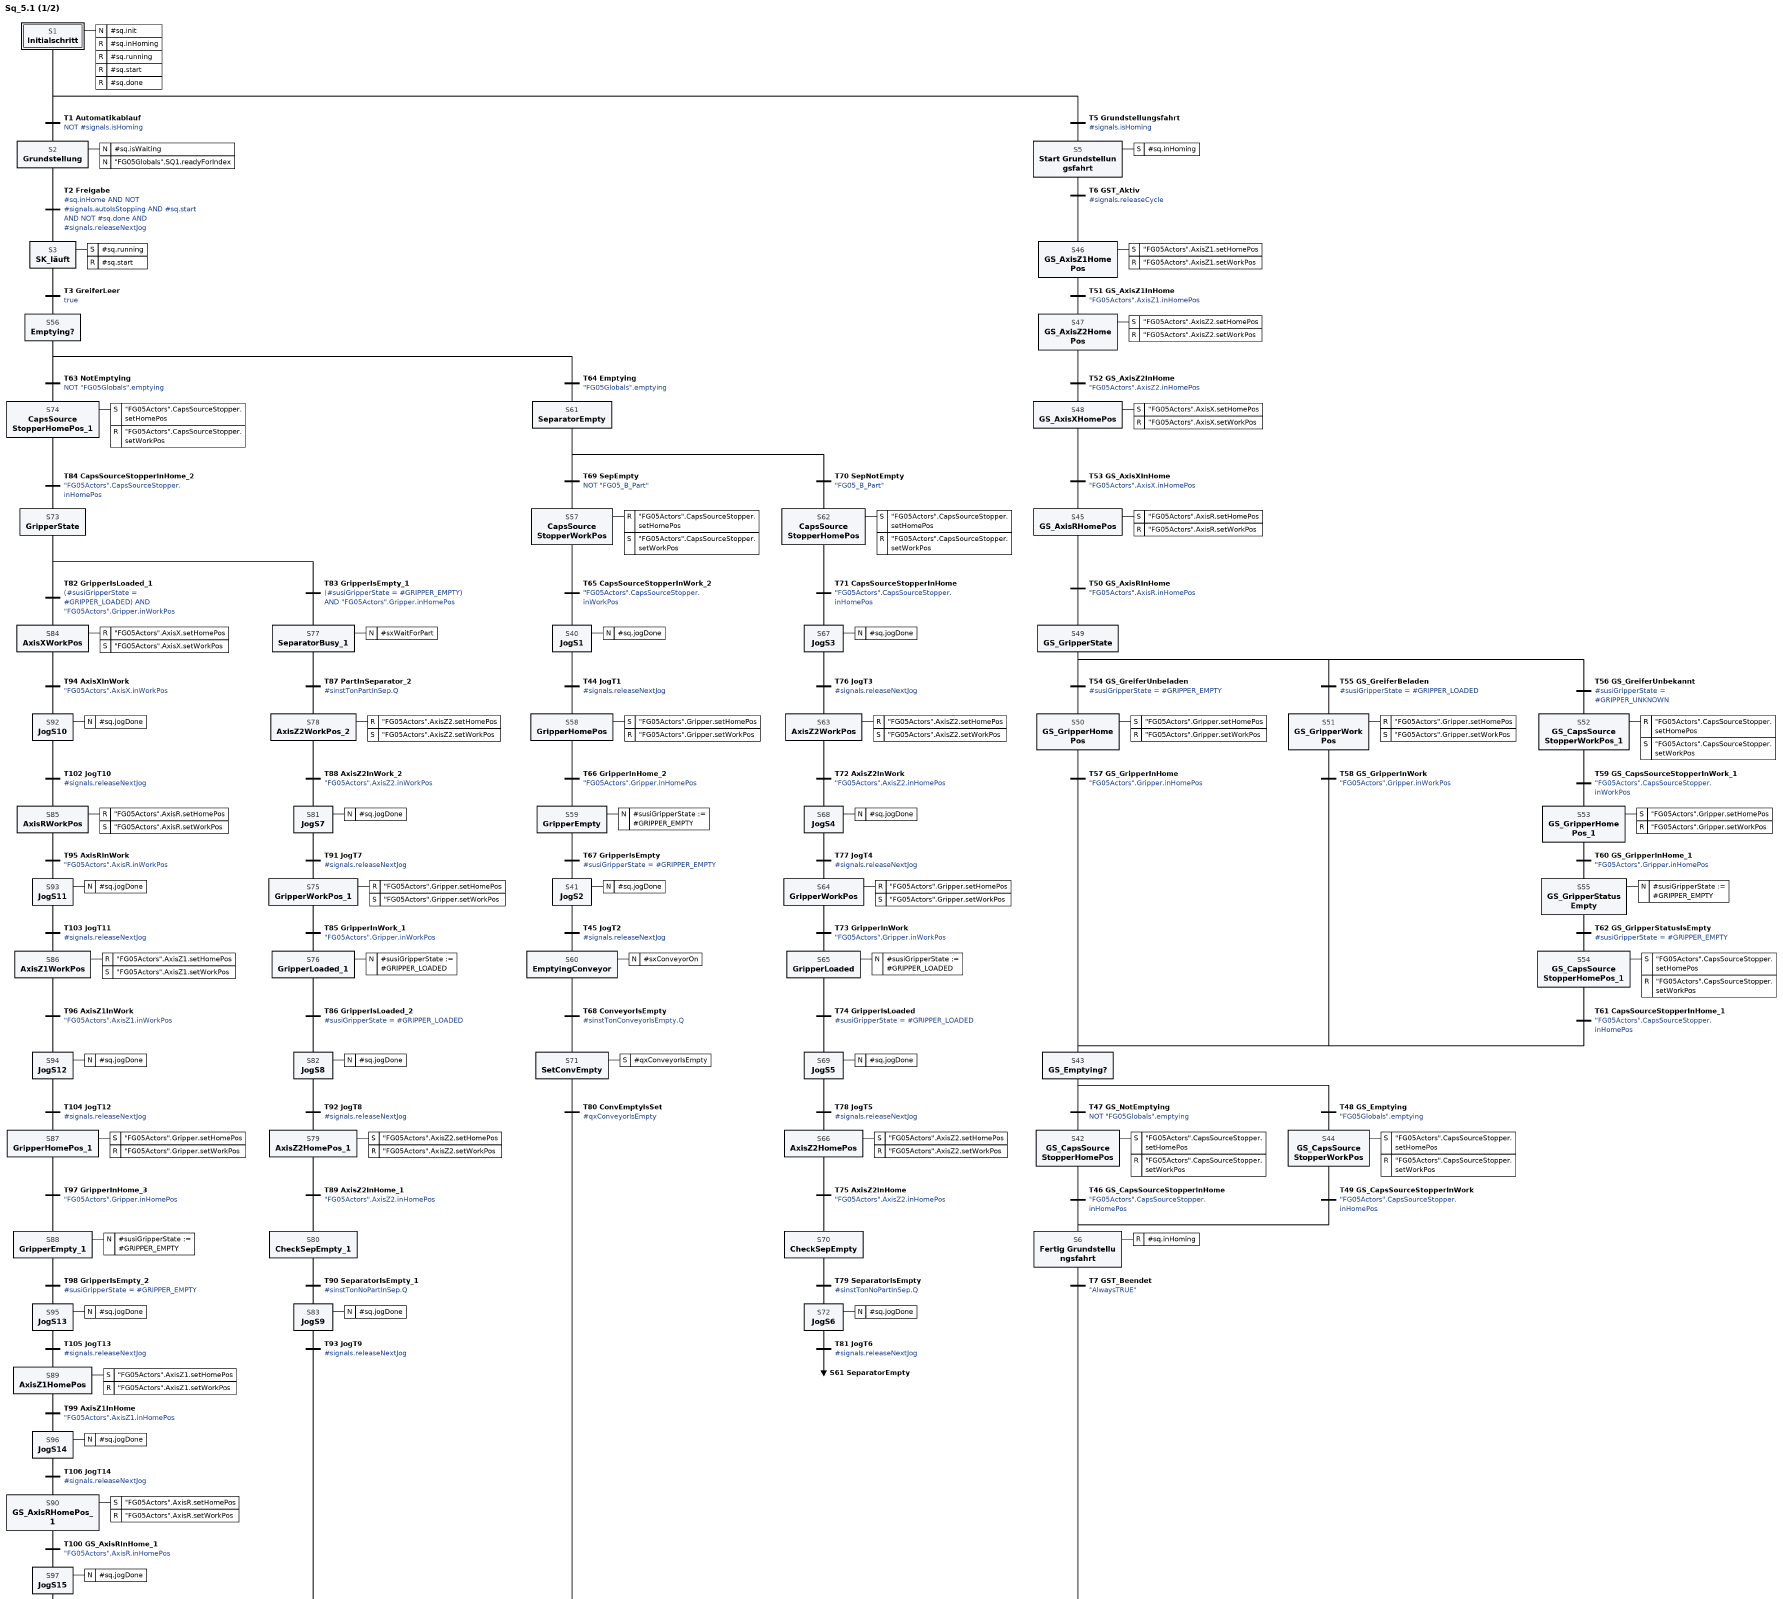
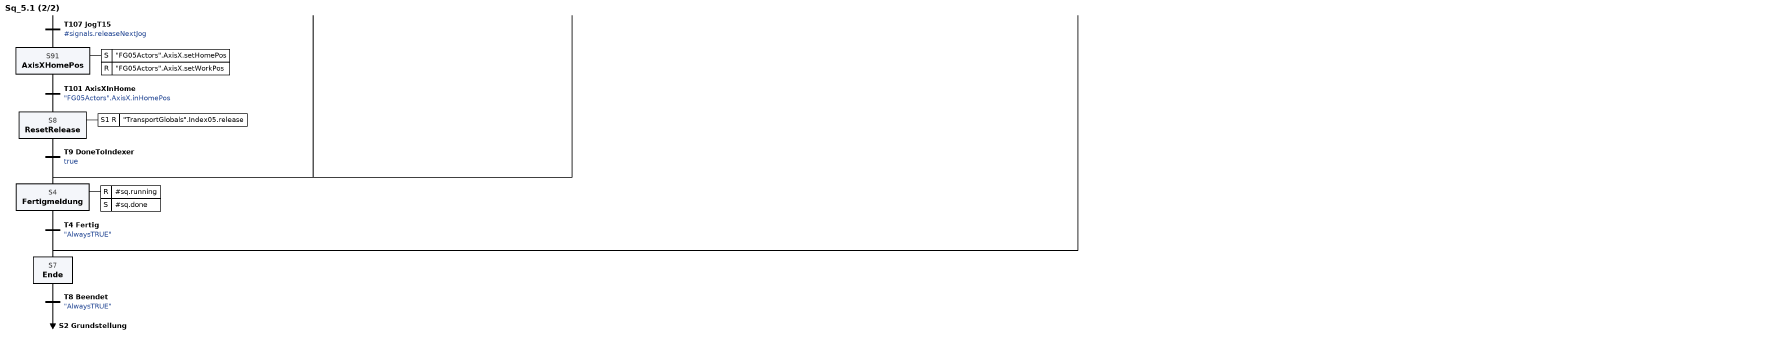
   // permanent pre-instructions
   NETWORK 1
   TITLE = Schrittkette verfügbar
      #sq.exists := true;
   NETWORK 2
   TITLE = Schrittkette in Grundstellung
      #sq.inHome := ("FG05Actors".CapsSourceStopper.inHomePos OR "FG05Actors".CapsSourceStopper.inWorkPos) AND (((#susiGripperState = #GRIPPER_EMPTY) AND "FG05Actors".Gripper.inHomePos) OR ((#susiGripperState = #GRIPPER_LOADED) AND "FG05Actors".Gripper.inWorkPos)) AND #Grundstellung.X AND "FG05Actors".AxisR.inHomePos AND "FG05Actors".AxisX.inHomePos AND "FG05Actors".AxisZ1.inHomePos AND "FG05Actors".AxisZ2.inHomePos;
   NETWORK 3
   TITLE = Startbedingung (Erweitern)
      #txStartCondition := ((((#susiGripperState = #GRIPPER_EMPTY) AND "FG05Actors".Gripper.inHomePos) OR "TransportGlobals".Index05.release) AND NOT "FG05Globals".emptying) OR ("FG05Globals".emptying AND NOT #qxConveyorIsEmpty);
   NETWORK 4
   TITLE = Schrittkette starten
      IF #sq.inHome AND NOT #sq.running AND #signals.releaseCycle AND NOT #signals.isHoming AND #txStartCondition THEN
          #sq.start := TRUE;
          #sq.done := FALSE;
      END_IF;
   NETWORK 5
   TITLE = ReleaseCycle Timer
      // ENO of a box is taken as its EN; it also drops when the box reports an error
      #_w1 := #ERR_FLT AND #ACK_EF;
      #_w2 := #_w1 AND NOT #sstReleaseCycle.ErrorAck;   // rising edge
      #sstReleaseCycle.ErrorAck := #_w1;
      IF (#S_NO <> #sstReleaseCycle.No_LastCycle) OR #_w2 THEN
          #sstReleaseCycle.T := T#0MS;
          #sstReleaseCycle.TckPrev := #sstReleaseCycle.Tck;
          #sstReleaseCycle.No_LastCycle := #S_NO;
      END_IF;
      #sstReleaseCycle.Tck := TIME_TCK();
      #tdTckDiff := #sstReleaseCycle.Tck - #sstReleaseCycle.TckPrev;
      #sstReleaseCycle.TckPrev := #sstReleaseCycle.Tck;
      IF (0 <= #tdTckDiff) AND (#tdTckDiff <= 1000) AND #signals.releaseCycle THEN
          #sstReleaseCycle.T := #sstReleaseCycle.T + #tdTckDiff;
      END_IF;

   // sequencer 1
   INITIAL_STEP Initialschritt:   // S1, max time T#10S, warning time T#7S
              N    #sq.init
              R    #sq.inHoming
              R    #sq.running
              R    #sq.start
              R    #sq.done
   END_STEP
   TRANSITION Automatikablauf FROM Initialschritt TO Grundstellung   // T1
      := NOT #signals.isHoming;
   END_TRANSITION
   TRANSITION Grundstellungsfahrt FROM Initialschritt TO "Start Grundstellungsfahrt"   // T5
      := #signals.isHoming;
   END_TRANSITION
   STEP Grundstellung:   // S2, max time T#10S, warning time T#7S
      supervision V := (#Grundstellung.U > t#5S) AND NOT #sq.inHome AND #signals.releaseCycle;
              N    #sq.isWaiting
              N    "FG05Globals".SQ1.readyForIndex
   END_STEP
   TRANSITION Freigabe FROM Grundstellung TO SK_läuft   // T2
      := #sq.inHome AND NOT #signals.autoIsStopping AND #sq.start AND NOT #sq.done AND #signals.releaseNextJog;
   END_TRANSITION
   STEP SK_läuft:   // S3, max time T#10S, warning time T#7S
              S    #sq.running
              R    #sq.start
   END_STEP
   TRANSITION GreiferLeer FROM SK_läuft TO "Emptying?"   // T3
      := true;
   END_TRANSITION
   STEP Fertigmeldung:   // S4, max time T#10S, warning time T#7S
              R    #sq.running
              S    #sq.done
   END_STEP
   TRANSITION Fertig FROM Fertigmeldung TO Ende   // T4
      := "AlwaysTRUE";
   END_TRANSITION
   STEP "Start Grundstellungsfahrt":   // S5, max time T#10S, warning time T#7S
              S    #sq.inHoming
   END_STEP
   TRANSITION GST_Aktiv FROM "Start Grundstellungsfahrt" TO GS_AxisZ1HomePos   // T6
      := #signals.releaseCycle;
   END_TRANSITION
   STEP "Fertig Grundstellungsfahrt":   // S6, max time T#10S, warning time T#7S
              R    #sq.inHoming
   END_STEP
   TRANSITION GST_Beendet FROM "Fertig Grundstellungsfahrt" TO Ende   // T7
      := "AlwaysTRUE";
   END_TRANSITION
   STEP Ende:   // S7, max time T#10S, warning time T#7S
   END_STEP
   TRANSITION Beendet FROM Ende TO Grundstellung   // T8, jump
      := "AlwaysTRUE";
   END_TRANSITION
   STEP JogS1:   // S40, max time T#10S, warning time T#7S
              N    #sq.jogDone
   END_STEP
   TRANSITION JogT1 FROM JogS1 TO GripperHomePos   // T44
      := #signals.releaseNextJog;
   END_TRANSITION
   STEP ResetRelease:   // S8, max time T#10S, warning time T#7S
      supervision V := (#ResetRelease.U >= t#10s) AND NOT #DoneToIndexer.TT AND #signals.releaseCycle;
          S1  R    "TransportGlobals".Index05.release
   END_STEP
   TRANSITION DoneToIndexer FROM ResetRelease TO Fertigmeldung   // T9
      := true;
   END_TRANSITION
   STEP CapsSourceStopperWorkPos:   // S57, max time T#10S, warning time T#7S
      supervision V := #sstReleaseCycle.T >= #itMaxRuntime;
              R    "FG05Actors".CapsSourceStopper.setHomePos
              S    "FG05Actors".CapsSourceStopper.setWorkPos
   END_STEP
   TRANSITION CapsSourceStopperInWork_2 FROM CapsSourceStopperWorkPos TO JogS1   // T65
      := "FG05Actors".CapsSourceStopper.inWorkPos;
   END_TRANSITION
   STEP "Emptying?":   // S56, max time T#10S, warning time T#7S
   END_STEP
   TRANSITION NotEmptying FROM "Emptying?" TO CapsSourceStopperHomePos_1   // T63
      := NOT "FG05Globals".emptying;
   END_TRANSITION
   TRANSITION Emptying FROM "Emptying?" TO SeparatorEmpty   // T64
      := "FG05Globals".emptying;
   END_TRANSITION
   STEP AxisRWorkPos:   // S85, max time T#10S, warning time T#7S
      supervision V := #sstReleaseCycle.T >= #itMaxRuntime;
              R    "FG05Actors".AxisR.setHomePos
              S    "FG05Actors".AxisR.setWorkPos
   END_STEP
   TRANSITION AxisRInWork FROM AxisRWorkPos TO JogS11   // T95
      := "FG05Actors".AxisR.inWorkPos;
   END_TRANSITION
   STEP "GS_Emptying?":   // S43, max time T#10S, warning time T#7S
   END_STEP
   TRANSITION GS_NotEmptying FROM "GS_Emptying?" TO GS_CapsSourceStopperHomePos   // T47
      := NOT "FG05Globals".emptying;
   END_TRANSITION
   TRANSITION GS_Emptying FROM "GS_Emptying?" TO GS_CapsSourceStopperWorkPos   // T48
      := "FG05Globals".emptying;
   END_TRANSITION
   STEP GS_CapsSourceStopperHomePos:   // S42, max time T#10S, warning time T#7S
      supervision V := #sstReleaseCycle.T >= #itMaxRuntime;
              S    "FG05Actors".CapsSourceStopper.setHomePos
              R    "FG05Actors".CapsSourceStopper.setWorkPos
   END_STEP
   TRANSITION GS_CapsSourceStopperInHome FROM GS_CapsSourceStopperHomePos TO "Fertig Grundstellungsfahrt"   // T46
      := "FG05Actors".CapsSourceStopper.inHomePos;
   END_TRANSITION
   STEP GS_CapsSourceStopperWorkPos:   // S44, max time T#10S, warning time T#7S
      supervision V := #sstReleaseCycle.T >= #itMaxRuntime;
              S    "FG05Actors".CapsSourceStopper.setHomePos
              R    "FG05Actors".CapsSourceStopper.setWorkPos
   END_STEP
   TRANSITION GS_CapsSourceStopperInWork FROM GS_CapsSourceStopperWorkPos TO "Fertig Grundstellungsfahrt"   // T49
      := "FG05Actors".CapsSourceStopper.inHomePos;
   END_TRANSITION
   STEP GS_AxisRHomePos:   // S45, max time T#10S, warning time T#7S
      supervision V := #sstReleaseCycle.T >= #itMaxRuntime;
              S    "FG05Actors".AxisR.setHomePos
              R    "FG05Actors".AxisR.setWorkPos
   END_STEP
   TRANSITION GS_AxisRInHome FROM GS_AxisRHomePos TO GS_GripperState   // T50
      := "FG05Actors".AxisR.inHomePos;
   END_TRANSITION
   STEP GS_AxisZ1HomePos:   // S46, max time T#10S, warning time T#7S
      supervision V := #sstReleaseCycle.T >= #itMaxRuntime;
              S    "FG05Actors".AxisZ1.setHomePos
              R    "FG05Actors".AxisZ1.setWorkPos
   END_STEP
   TRANSITION GS_AxisZ1InHome FROM GS_AxisZ1HomePos TO GS_AxisZ2HomePos   // T51
      := "FG05Actors".AxisZ1.inHomePos;
   END_TRANSITION
   STEP GS_AxisZ2HomePos:   // S47, max time T#10S, warning time T#7S
      supervision V := #sstReleaseCycle.T >= #itMaxRuntime;
              S    "FG05Actors".AxisZ2.setHomePos
              R    "FG05Actors".AxisZ2.setWorkPos
   END_STEP
   TRANSITION GS_AxisZ2InHome FROM GS_AxisZ2HomePos TO GS_AxisXHomePos   // T52
      := "FG05Actors".AxisZ2.inHomePos;
   END_TRANSITION
   STEP GS_AxisXHomePos:   // S48, max time T#10S, warning time T#7S
      supervision V := #sstReleaseCycle.T >= #itMaxRuntime;
              S    "FG05Actors".AxisX.setHomePos
              R    "FG05Actors".AxisX.setWorkPos
   END_STEP
   TRANSITION GS_AxisXInHome FROM GS_AxisXHomePos TO GS_AxisRHomePos   // T53
      := "FG05Actors".AxisX.inHomePos;
   END_TRANSITION
   STEP GS_GripperState:   // S49, max time T#10S, warning time T#7S
   END_STEP
   TRANSITION GS_GreiferUnbeladen FROM GS_GripperState TO GS_GripperHomePos   // T54
      := #susiGripperState = #GRIPPER_EMPTY;
   END_TRANSITION
   TRANSITION GS_GreiferBeladen FROM GS_GripperState TO GS_GripperWorkPos   // T55
      := #susiGripperState = #GRIPPER_LOADED;
   END_TRANSITION
   TRANSITION GS_GreiferUnbekannt FROM GS_GripperState TO GS_CapsSourceStopperWorkPos_1   // T56
      := #susiGripperState = #GRIPPER_UNKNOWN;
   END_TRANSITION
   STEP GS_GripperHomePos:   // S50, max time T#10S, warning time T#7S
      supervision V := #sstReleaseCycle.T >= #itMaxRuntime;
              S    "FG05Actors".Gripper.setHomePos
              R    "FG05Actors".Gripper.setWorkPos
   END_STEP
   TRANSITION GS_GripperInHome FROM GS_GripperHomePos TO "GS_Emptying?"   // T57
      := "FG05Actors".Gripper.inHomePos;
   END_TRANSITION
   STEP GS_GripperWorkPos:   // S51, max time T#10S, warning time T#7S
      supervision V := #sstReleaseCycle.T >= #itMaxRuntime;
              R    "FG05Actors".Gripper.setHomePos
              S    "FG05Actors".Gripper.setWorkPos
   END_STEP
   TRANSITION GS_GripperInWork FROM GS_GripperWorkPos TO "GS_Emptying?"   // T58
      := "FG05Actors".Gripper.inWorkPos;
   END_TRANSITION
   STEP GS_CapsSourceStopperWorkPos_1:   // S52, max time T#10S, warning time T#7S
      supervision V := #sstReleaseCycle.T >= #itMaxRuntime;
              R    "FG05Actors".CapsSourceStopper.setHomePos
              S    "FG05Actors".CapsSourceStopper.setWorkPos
   END_STEP
   TRANSITION GS_CapsSourceStopperInWork_1 FROM GS_CapsSourceStopperWorkPos_1 TO GS_GripperHomePos_1   // T59
      := "FG05Actors".CapsSourceStopper.inWorkPos;
   END_TRANSITION
   STEP GS_GripperHomePos_1:   // S53, max time T#10S, warning time T#7S
      supervision V := #sstReleaseCycle.T >= #itMaxRuntime;
              S    "FG05Actors".Gripper.setHomePos
              R    "FG05Actors".Gripper.setWorkPos
   END_STEP
   TRANSITION GS_GripperInHome_1 FROM GS_GripperHomePos_1 TO GS_GripperStatusEmpty   // T60
      := "FG05Actors".Gripper.inHomePos;
   END_TRANSITION
   STEP GS_CapsSourceStopperHomePos_1:   // S54, max time T#10S, warning time T#7S
      supervision V := #sstReleaseCycle.T >= #itMaxRuntime;
              S    "FG05Actors".CapsSourceStopper.setHomePos
              R    "FG05Actors".CapsSourceStopper.setWorkPos
   END_STEP
   TRANSITION CapsSourceStopperInHome_1 FROM GS_CapsSourceStopperHomePos_1 TO "GS_Emptying?"   // T61
      := "FG05Actors".CapsSourceStopper.inHomePos;
   END_TRANSITION
   STEP GS_GripperStatusEmpty:   // S55, max time T#10S, warning time T#7S
              N    #susiGripperState := #GRIPPER_EMPTY
   END_STEP
   TRANSITION GS_GripperStatusIsEmpty FROM GS_GripperStatusEmpty TO GS_CapsSourceStopperHomePos_1   // T62
      := #susiGripperState = #GRIPPER_EMPTY;
   END_TRANSITION
   STEP GripperHomePos:   // S58, max time T#10S, warning time T#7S
      supervision V := #sstReleaseCycle.T >= #itMaxRuntime;
              S    "FG05Actors".Gripper.setHomePos
              R    "FG05Actors".Gripper.setWorkPos
   END_STEP
   TRANSITION GripperInHome_2 FROM GripperHomePos TO GripperEmpty   // T66
      := "FG05Actors".Gripper.inHomePos;
   END_TRANSITION
   STEP GripperEmpty:   // S59, max time T#10S, warning time T#7S
              N    #susiGripperState := #GRIPPER_EMPTY
   END_STEP
   TRANSITION GripperIsEmpty FROM GripperEmpty TO JogS2   // T67
      := #susiGripperState = #GRIPPER_EMPTY;
   END_TRANSITION
   STEP JogS2:   // S41, max time T#10S, warning time T#7S
              N    #sq.jogDone
   END_STEP
   TRANSITION JogT2 FROM JogS2 TO EmptyingConveyor   // T45
      := #signals.releaseNextJog;
   END_TRANSITION
   STEP EmptyingConveyor:   // S60, max time T#10S, warning time T#7S
              N    #sxConveyorOn
   END_STEP
   TRANSITION ConveyorIsEmpty FROM EmptyingConveyor TO SetConvEmpty   // T68
      := #sinstTonConveyorIsEmpty.Q;
   END_TRANSITION
   STEP SeparatorEmpty:   // S61, max time T#10S, warning time T#7S
   END_STEP
   TRANSITION SepEmpty FROM SeparatorEmpty TO CapsSourceStopperWorkPos   // T69
      := NOT "FG05_B_Part";
   END_TRANSITION
   TRANSITION SepNotEmpty FROM SeparatorEmpty TO CapsSourceStopperHomePos   // T70
      := "FG05_B_Part";
   END_TRANSITION
   STEP CapsSourceStopperHomePos:   // S62, max time T#10S, warning time T#7S
      supervision V := #sstReleaseCycle.T >= #itMaxRuntime;
              S    "FG05Actors".CapsSourceStopper.setHomePos
              R    "FG05Actors".CapsSourceStopper.setWorkPos
   END_STEP
   TRANSITION CapsSourceStopperInHome FROM CapsSourceStopperHomePos TO JogS3   // T71
      := "FG05Actors".CapsSourceStopper.inHomePos;
   END_TRANSITION
   STEP AxisZ2WorkPos:   // S63, max time T#10S, warning time T#7S
      supervision V := #sstReleaseCycle.T >= #itMaxRuntime;
              R    "FG05Actors".AxisZ2.setHomePos
              S    "FG05Actors".AxisZ2.setWorkPos
   END_STEP
   TRANSITION AxisZ2InWork FROM AxisZ2WorkPos TO JogS4   // T72
      := "FG05Actors".AxisZ2.inHomePos;
   END_TRANSITION
   STEP GripperWorkPos:   // S64, max time T#10S, warning time T#7S
      supervision V := #sstReleaseCycle.T >= #itMaxRuntime;
              R    "FG05Actors".Gripper.setHomePos
              S    "FG05Actors".Gripper.setWorkPos
   END_STEP
   TRANSITION GripperInWork FROM GripperWorkPos TO GripperLoaded   // T73
      := "FG05Actors".Gripper.inWorkPos;
   END_TRANSITION
   STEP GripperLoaded:   // S65, max time T#10S, warning time T#7S
              N    #susiGripperState := #GRIPPER_LOADED
   END_STEP
   TRANSITION GripperIsLoaded FROM GripperLoaded TO JogS5   // T74
      := #susiGripperState = #GRIPPER_LOADED;
   END_TRANSITION
   STEP AxisZ2HomePos:   // S66, max time T#10S, warning time T#7S
      supervision V := #sstReleaseCycle.T >= #itMaxRuntime;
              S    "FG05Actors".AxisZ2.setHomePos
              R    "FG05Actors".AxisZ2.setWorkPos
   END_STEP
   TRANSITION AxisZ2InHome FROM AxisZ2HomePos TO CheckSepEmpty   // T75
      := "FG05Actors".AxisZ2.inHomePos;
   END_TRANSITION
   STEP CheckSepEmpty:   // S70, max time T#10S, warning time T#7S
      supervision V := #sstReleaseCycle.T >= #itMaxRuntime;
   END_STEP
   TRANSITION SeparatorIsEmpty FROM CheckSepEmpty TO JogS6   // T79
      := #sinstTonNoPartInSep.Q;
   END_TRANSITION
   STEP SetConvEmpty:   // S71, max time T#10S, warning time T#7S
              S    #qxConveyorIsEmpty
   END_STEP
   TRANSITION ConvEmptyIsSet FROM SetConvEmpty TO Fertigmeldung   // T80
      := #qxConveyorIsEmpty;
   END_TRANSITION
   STEP JogS3:   // S67, max time T#10S, warning time T#7S
              N    #sq.jogDone
   END_STEP
   TRANSITION JogT3 FROM JogS3 TO AxisZ2WorkPos   // T76
      := #signals.releaseNextJog;
   END_TRANSITION
   STEP JogS4:   // S68, max time T#10S, warning time T#7S
              N    #sq.jogDone
   END_STEP
   TRANSITION JogT4 FROM JogS4 TO GripperWorkPos   // T77
      := #signals.releaseNextJog;
   END_TRANSITION
   STEP JogS5:   // S69, max time T#10S, warning time T#7S
              N    #sq.jogDone
   END_STEP
   TRANSITION JogT5 FROM JogS5 TO AxisZ2HomePos   // T78
      := #signals.releaseNextJog;
   END_TRANSITION
   STEP JogS6:   // S72, max time T#10S, warning time T#7S
              N    #sq.jogDone
   END_STEP
   TRANSITION JogT6 FROM JogS6 TO SeparatorEmpty   // T81, jump
      := #signals.releaseNextJog;
   END_TRANSITION
   STEP GripperState:   // S73, max time T#10S, warning time T#7S
      supervision V := #sstReleaseCycle.T >= #itMaxRuntime;
   END_STEP
   TRANSITION GripperIsLoaded_1 FROM GripperState TO AxisXWorkPos   // T82
      := (#susiGripperState = #GRIPPER_LOADED) AND "FG05Actors".Gripper.inWorkPos;
   END_TRANSITION
   TRANSITION GripperIsEmpty_1 FROM GripperState TO SeparatorBusy_1   // T83
      := (#susiGripperState = #GRIPPER_EMPTY) AND "FG05Actors".Gripper.inHomePos;
   END_TRANSITION
   STEP CapsSourceStopperHomePos_1:   // S74, max time T#10S, warning time T#7S
      supervision V := #sstReleaseCycle.T >= #itMaxRuntime;
              S    "FG05Actors".CapsSourceStopper.setHomePos
              R    "FG05Actors".CapsSourceStopper.setWorkPos
   END_STEP
   TRANSITION CapsSourceStopperInHome_2 FROM CapsSourceStopperHomePos_1 TO GripperState   // T84
      := "FG05Actors".CapsSourceStopper.inHomePos;
   END_TRANSITION
   STEP GripperWorkPos_1:   // S75, max time T#10S, warning time T#7S
      supervision V := #sstReleaseCycle.T >= #itMaxRuntime;
              R    "FG05Actors".Gripper.setHomePos
              S    "FG05Actors".Gripper.setWorkPos
   END_STEP
   TRANSITION GripperInWork_1 FROM GripperWorkPos_1 TO GripperLoaded_1   // T85
      := "FG05Actors".Gripper.inWorkPos;
   END_TRANSITION
   STEP GripperLoaded_1:   // S76, max time T#10S, warning time T#7S
              N    #susiGripperState := #GRIPPER_LOADED
   END_STEP
   TRANSITION GripperIsLoaded_2 FROM GripperLoaded_1 TO JogS8   // T86
      := #susiGripperState = #GRIPPER_LOADED;
   END_TRANSITION
   STEP SeparatorBusy_1:   // S77, max time T#10S, warning time T#7S
              N    #sxWaitForPart
   END_STEP
   TRANSITION PartInSeparator_2 FROM SeparatorBusy_1 TO AxisZ2WorkPos_2   // T87
      := #sinstTonPartInSep.Q;
   END_TRANSITION
   STEP AxisZ2WorkPos_2:   // S78, max time T#10S, warning time T#7S
      supervision V := #sstReleaseCycle.T >= #itMaxRuntime;
              R    "FG05Actors".AxisZ2.setHomePos
              S    "FG05Actors".AxisZ2.setWorkPos
   END_STEP
   TRANSITION AxisZ2InWork_2 FROM AxisZ2WorkPos_2 TO JogS7   // T88
      := "FG05Actors".AxisZ2.inWorkPos;
   END_TRANSITION
   STEP AxisZ2HomePos_1:   // S79, max time T#10S, warning time T#7S
      supervision V := #sstReleaseCycle.T >= #itMaxRuntime;
              S    "FG05Actors".AxisZ2.setHomePos
              R    "FG05Actors".AxisZ2.setWorkPos
   END_STEP
   TRANSITION AxisZ2InHome_1 FROM AxisZ2HomePos_1 TO CheckSepEmpty_1   // T89
      := "FG05Actors".AxisZ2.inHomePos;
   END_TRANSITION
   STEP CheckSepEmpty_1:   // S80, max time T#10S, warning time T#7S
      supervision V := #sstReleaseCycle.T >= #itMaxRuntime;
   END_STEP
   TRANSITION SeparatorIsEmpty_1 FROM CheckSepEmpty_1 TO JogS9   // T90
      := #sinstTonNoPartInSep.Q;
   END_TRANSITION
   STEP JogS7:   // S81, max time T#10S, warning time T#7S
              N    #sq.jogDone
   END_STEP
   TRANSITION JogT7 FROM JogS7 TO GripperWorkPos_1   // T91
      := #signals.releaseNextJog;
   END_TRANSITION
   STEP JogS8:   // S82, max time T#10S, warning time T#7S
              N    #sq.jogDone
   END_STEP
   TRANSITION JogT8 FROM JogS8 TO AxisZ2HomePos_1   // T92
      := #signals.releaseNextJog;
   END_TRANSITION
   STEP JogS9:   // S83, max time T#10S, warning time T#7S
              N    #sq.jogDone
   END_STEP
   TRANSITION JogT9 FROM JogS9 TO Fertigmeldung   // T93
      := #signals.releaseNextJog;
   END_TRANSITION
   STEP AxisXWorkPos:   // S84, max time T#10S, warning time T#7S
      supervision V := #sstReleaseCycle.T >= #itMaxRuntime;
              R    "FG05Actors".AxisX.setHomePos
              S    "FG05Actors".AxisX.setWorkPos
   END_STEP
   TRANSITION AxisXInWork FROM AxisXWorkPos TO JogS10   // T94
      := "FG05Actors".AxisX.inWorkPos;
   END_TRANSITION
   STEP AxisZ1WorkPos:   // S86, max time T#10S, warning time T#7S
      supervision V := #sstReleaseCycle.T >= #itMaxRuntime;
              R    "FG05Actors".AxisZ1.setHomePos
              S    "FG05Actors".AxisZ1.setWorkPos
   END_STEP
   TRANSITION AxisZ1InWork FROM AxisZ1WorkPos TO JogS12   // T96
      := "FG05Actors".AxisZ1.inWorkPos;
   END_TRANSITION
   STEP GripperHomePos_1:   // S87, max time T#10S, warning time T#7S
      supervision V := #sstReleaseCycle.T >= #itMaxRuntime;
              S    "FG05Actors".Gripper.setHomePos
              R    "FG05Actors".Gripper.setWorkPos
   END_STEP
   TRANSITION GripperInHome_3 FROM GripperHomePos_1 TO GripperEmpty_1   // T97
      := "FG05Actors".Gripper.inHomePos;
   END_TRANSITION
   STEP GripperEmpty_1:   // S88, max time T#10S, warning time T#7S
              N    #susiGripperState := #GRIPPER_EMPTY
   END_STEP
   TRANSITION GripperIsEmpty_2 FROM GripperEmpty_1 TO JogS13   // T98
      := #susiGripperState = #GRIPPER_EMPTY;
   END_TRANSITION
   STEP AxisZ1HomePos:   // S89, max time T#10S, warning time T#7S
      supervision V := #sstReleaseCycle.T >= #itMaxRuntime;
              S    "FG05Actors".AxisZ1.setHomePos
              R    "FG05Actors".AxisZ1.setWorkPos
   END_STEP
   TRANSITION AxisZ1InHome FROM AxisZ1HomePos TO JogS14   // T99
      := "FG05Actors".AxisZ1.inHomePos;
   END_TRANSITION
   STEP GS_AxisRHomePos_1:   // S90, max time T#10S, warning time T#7S
      supervision V := #sstReleaseCycle.T >= #itMaxRuntime;
              S    "FG05Actors".AxisR.setHomePos
              R    "FG05Actors".AxisR.setWorkPos
   END_STEP
   TRANSITION GS_AxisRInHome_1 FROM GS_AxisRHomePos_1 TO JogS15   // T100
      := "FG05Actors".AxisR.inHomePos;
   END_TRANSITION
   STEP AxisXHomePos:   // S91, max time T#10S, warning time T#7S
      supervision V := #sstReleaseCycle.T >= #itMaxRuntime;
              S    "FG05Actors".AxisX.setHomePos
              R    "FG05Actors".AxisX.setWorkPos
   END_STEP
   TRANSITION AxisXInHome FROM AxisXHomePos TO ResetRelease   // T101
      := "FG05Actors".AxisX.inHomePos;
   END_TRANSITION
   STEP JogS10:   // S92, max time T#10S, warning time T#7S
              N    #sq.jogDone
   END_STEP
   TRANSITION JogT10 FROM JogS10 TO AxisRWorkPos   // T102
      := #signals.releaseNextJog;
   END_TRANSITION
   STEP JogS11:   // S93, max time T#10S, warning time T#7S
              N    #sq.jogDone
   END_STEP
   TRANSITION JogT11 FROM JogS11 TO AxisZ1WorkPos   // T103
      := #signals.releaseNextJog;
   END_TRANSITION
   STEP JogS12:   // S94, max time T#10S, warning time T#7S
              N    #sq.jogDone
   END_STEP
   TRANSITION JogT12 FROM JogS12 TO GripperHomePos_1   // T104
      := #signals.releaseNextJog;
   END_TRANSITION
   STEP JogS13:   // S95, max time T#10S, warning time T#7S
              N    #sq.jogDone
   END_STEP
   TRANSITION JogT13 FROM JogS13 TO AxisZ1HomePos   // T105
      := #signals.releaseNextJog;
   END_TRANSITION
   STEP JogS14:   // S96, max time T#10S, warning time T#7S
              N    #sq.jogDone
   END_STEP
   TRANSITION JogT14 FROM JogS14 TO GS_AxisRHomePos_1   // T106
      := #signals.releaseNextJog;
   END_TRANSITION
   STEP JogS15:   // S97, max time T#10S, warning time T#7S
              N    #sq.jogDone
   END_STEP
   TRANSITION JogT15 FROM JogS15 TO AxisXHomePos   // T107
      := #signals.releaseNextJog;
   END_TRANSITION

   // permanent post-instructions
   NETWORK 1
   TITLE = Störungssignal weitergeben
      #sq.error := #ERR_FLT;
   NETWORK 2
   TITLE = Ablauf ist aktiv
      #qxIsActive := #sq.running;
   NETWORK 3
   TITLE = steht in Grundstellung
      #qxIsInHome := #sq.inHome AND NOT #sq.running;
   NETWORK 4
   TITLE = wenn Einrichten aktiv war, ist Greiferzustand unbekannt
      IF #signals.setupActive THEN #susiGripperState := #GRIPPER_UNKNOWN; END_IF;
   NETWORK 5
   TITLE = Bunker einschalten
      "FG05Actors".Bunker.setWorkPos := "FG05Actors".Conveyor.workAct AND NOT "FG05Globals".emptying;
   NETWORK 6
   TITLE = Conveyor einschalten
      #sinstTofConveyorOn(IN := #signals.releaseCycle, PT := t#30s);   // TOF
      "FG05Actors".Conveyor.setWorkPos := (#sinstTofConveyorOn.Q AND "FG05Actors".CapsSourceStopper.inHomePos AND NOT #signals.isHoming AND NOT "FG05Globals".emptying) OR (#sxConveyorOn AND "FG05Globals".emptying);
   NETWORK 7
   TITLE = Conveyor ist leer
      IF "FG05_B_Part" OR NOT "FG05Globals".emptying THEN #qxConveyorIsEmpty := FALSE; END_IF;
      #sinstTonConveyorIsEmpty(IN := NOT "FG05_B_Part" AND "FG05Actors".Conveyor.setWorkPos, PT := t#20s);   // TON
   NETWORK 8
   TITLE = Teil in der Vereinzelung
      #sinstTonPartInSep(IN := "FG05_B_Part", PT := t#250ms);   // TON
   NETWORK 9
   TITLE = Kein Teil in der Vereinzelung
      #sinstTonNoPartInSep(IN := NOT "FG05_B_Part", PT := t#250ms);   // TON
   NETWORK 10
   TITLE = Teilemangel
      #sinstTonLackOfParts(IN := #sxWaitForPart, PT := t#5s);   // TON
      #qxLackOfParts := #sinstTonLackOfParts.Q;
END_FUNCTION_BLOCK

FUNCTION "StepSequencesSt.5" : Void   // FC1510, FBD
TITLE = Schrittkettensteuerung
{ S7_Optimized_Access := 'TRUE' }
VERSION : 0.1
// Ersteller: Andreas Fast Automation
// E-Mail: automation@fast-andreas.de
// 
// Projekt dient zu Demonstrationszwecken und frei genutzt werden.
// 
// Bausteinbeschreibung:
   VAR_IN_OUT
      station : "typeStation";
   END_VAR
   VAR_TEMP
      tempInit : Bool;
      tempAck : Bool;
      tempAuto : Bool;
      tempMan : Bool;
      tempTap : Bool;
      tempPush : Bool;
   END_VAR
BEGIN

REGION Network 1: Graph Parameter
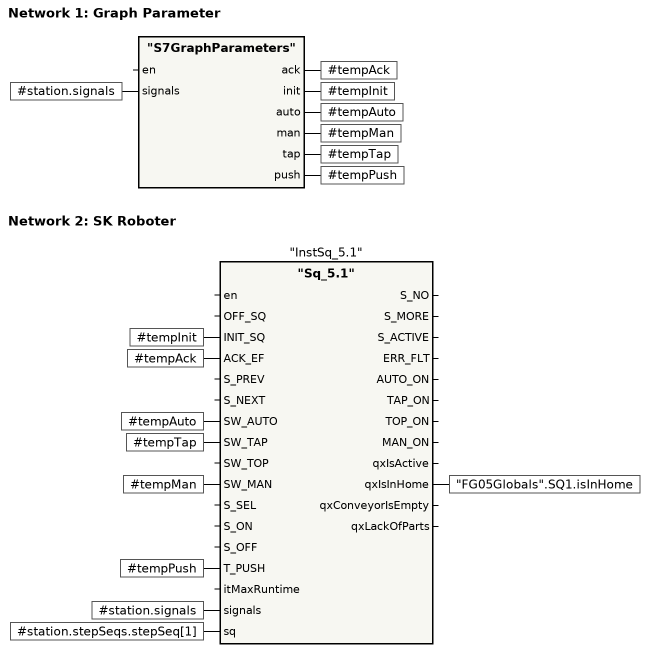
   "S7GraphParameters"(signals := #station.signals,
                       ack => #tempAck,
                       init => #tempInit,
                       auto => #tempAuto,
                       man => #tempMan,
                       tap => #tempTap,
                       push => #tempPush);
END_REGION

REGION Network 2: SK Roboter
   "InstSq_5.1"(INIT_SQ := #tempInit,   // "Sq_5.1"
                ACK_EF := #tempAck,
                SW_AUTO := #tempAuto,
                SW_TAP := #tempTap,
                SW_MAN := #tempMan,
                T_PUSH := #tempPush,
                signals := #station.signals,
                sq := #station.stepSeqs.stepSeq[1],
                qxIsInHome => "FG05Globals".SQ1.isInHome);
END_REGION
END_FUNCTION

// folder: 2. Machine/10_FG_Transport

FUNCTION_BLOCK "TransportControl"   // FB2000, FBD
TITLE = Station Transport Hauptaufruf
{ S7_Optimized_Access := 'TRUE' }
VERSION : 0.1
// Ersteller: Andreas Fast Automation
// E-Mail: automation@fast-andreas.de
// 
// Projekt dient zu Demonstrationszwecken und frei genutzt werden.
// 
// Bausteinbeschreibung:
   VAR_INPUT
      stationNo : Int := 10;   // Stationsnummer
   END_VAR
   VAR_IN_OUT
      machine : "typeMachine";
      station : "typeStation";
      manualMovement : "typeManualMovements";
      plcErrMsg : "typePlcErrMsg";
      hmiErrMsg : "typeHmiErrMsg";
   END_VAR
   VAR
      instStationControl : "StationControl";
      instActorControl : "TransportActorControl";
      sinstProcessStopper : "Process_Stopper";
      sinstTofRunConveyor1 : TOF_TIME;
      sinstTofRunConveyor2 : TOF_TIME;
   END_VAR
BEGIN

REGION Network 1: Stationssteuerung
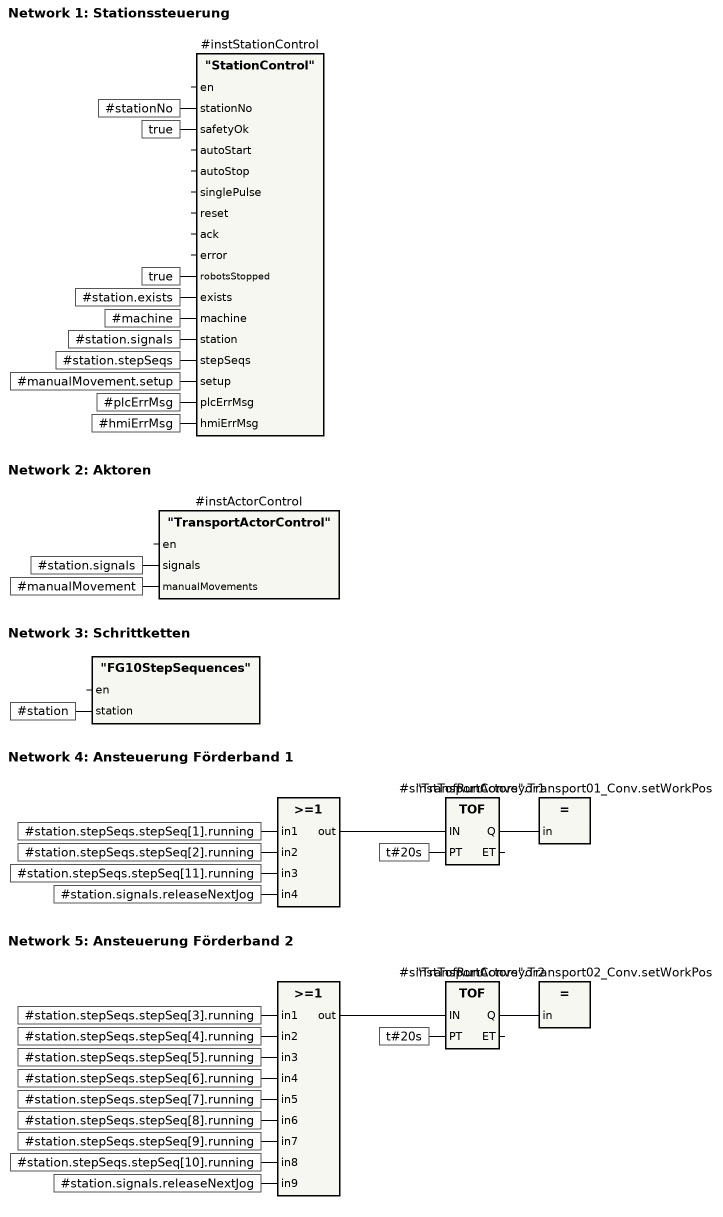
   #instStationControl(stationNo := #stationNo,   // "StationControl"
                       safetyOk := true,
                       robotsStopped := true,
                       exists := #station.exists,
                       machine := #machine,
                       station := #station.signals,
                       stepSeqs := #station.stepSeqs,
                       setup := #manualMovement.setup,
                       plcErrMsg := #plcErrMsg,
                       hmiErrMsg := #hmiErrMsg);
END_REGION

REGION Network 2: Aktoren
   #instActorControl(signals := #station.signals, manualMovements := #manualMovement);   // "TransportActorControl"
END_REGION

REGION Network 3: Schrittketten
   "FG10StepSequences"(station := #station);
END_REGION

REGION Network 4: Ansteuerung Förderband 1
   #sinstTofRunConveyor1(IN := #station.stepSeqs.stepSeq[1].running OR #station.stepSeqs.stepSeq[2].running OR #station.stepSeqs.stepSeq[11].running OR #station.signals.releaseNextJog,   // TOF
                         PT := t#20s);
   "TransportActors".Transport01_Conv.setWorkPos := #sinstTofRunConveyor1.Q;
END_REGION

REGION Network 5: Ansteuerung Förderband 2
   #sinstTofRunConveyor2(IN := #station.stepSeqs.stepSeq[3].running OR #station.stepSeqs.stepSeq[4].running OR #station.stepSeqs.stepSeq[5].running OR #station.stepSeqs.stepSeq[6].running OR #station.stepSeqs.stepSeq[7].running OR #station.stepSeqs.stepSeq[8].running OR #station.stepSeqs.stepSeq[9].running OR #station.stepSeqs.stepSeq[10].running OR #station.signals.releaseNextJog,   // TOF
                         PT := t#20s);
   "TransportActors".Transport02_Conv.setWorkPos := #sinstTofRunConveyor2.Q;
END_REGION
END_FUNCTION_BLOCK

FUNCTION_BLOCK "TransportActorControl"   // FB2002, FBD
TITLE = Aktoransteuerung
{ S7_Optimized_Access := 'TRUE' }
VERSION : 0.1
// Ersteller: Andreas Fast Automation
// E-Mail: automation@fast-andreas.de
// 
// Projekt dient zu Demonstrationszwecken und frei genutzt werden.
// 
// Bausteinbeschreibung:
   VAR_IN_OUT
      signals : "typeStationSignals";
      manualMovements : "typeManualMovements";
   END_VAR
   VAR
      instActorReserved1 : "Actor_Reserved";
      instActorReserved2 : "Actor_Reserved";
      instActorReserved3 : "Actor_Reserved";
      instActorReserved4 : "Actor_Reserved";
      instActorReserved5 : "Actor_Reserved";
      instActorReserved6 : "Actor_Reserved";
      sinstGate_1 : "Cylinder_1Out2In";
      sinstGate_2 : "Cylinder_1Out2In";
      sinstIndex01_Y_Lift : "Cylinder_2Out2In";
      sinstIndex01_Y_Stopper : "Cylinder_1Out1In (ungetestet)";
      sinstIndex02_Y_Lift : "Cylinder_2Out2In";
      sinstIndex02_Y_Stopper : "Cylinder_1Out1In (ungetestet)";
      sinstIndex03_Y_Lift : "Cylinder_2Out2In";
      sinstIndex03_Y_Stopper : "Cylinder_1Out1In (ungetestet)";
      sinstIndex04_Y_Lift : "Cylinder_2Out2In";
      sinstIndex04_Y_Stopper : "Cylinder_1Out1In (ungetestet)";
      sinstIndex05_Y_Lift : "Cylinder_2Out2In";
      sinstIndex05_Y_Stopper : "Cylinder_1Out1In (ungetestet)";
      sinstStopper01_Y_Stopper : "Cylinder_1Out1In (ungetestet)";
      sinstStopper02_Y_Stopper : "Cylinder_1Out1In (ungetestet)";
      sinstStopper03_Y_Stopper : "Cylinder_1Out1In (ungetestet)";
      sinstStopper04_Y_Stopper : "Cylinder_1Out1In (ungetestet)";
      sinstLift01_Y_Lift : "Cylinder_2Out2In";
      sinstLift01_M_Conveyor : "Motor_2Out";
      sinstLift02_Y_Lift : "Cylinder_2Out2In";
      sinstLift02_M_Conveyor : "Motor_2Out";
      sinstTransport01_M_Conveyor : "Motor_2Out";
      sinstTransport02_M_Conveyor : "Motor_2Out";
   END_VAR
BEGIN

REGION Network 1: Gate 1
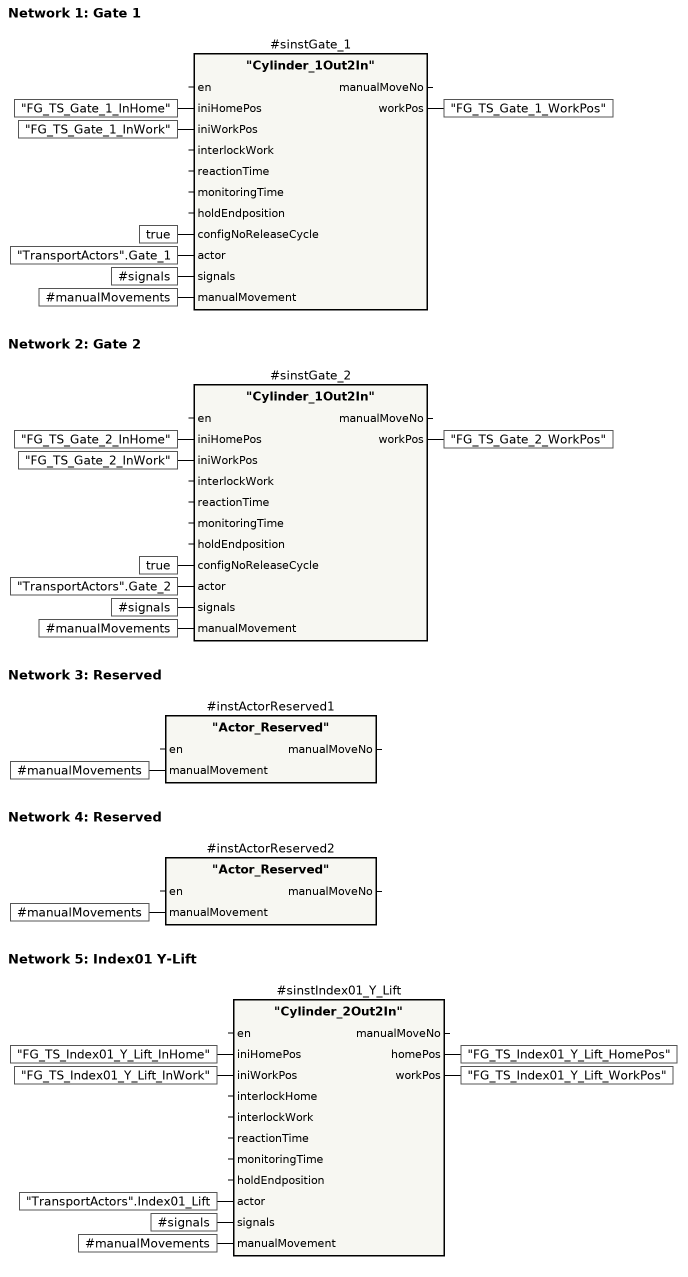
   #sinstGate_1(iniHomePos := "FG_TS_Gate_1_InHome",   // "Cylinder_1Out2In"
                iniWorkPos := "FG_TS_Gate_1_InWork",
                configNoReleaseCycle := true,
                actor := "TransportActors".Gate_1,
                signals := #signals,
                manualMovement := #manualMovements,
                workPos => "FG_TS_Gate_1_WorkPos");
END_REGION

REGION Network 2: Gate 2
   #sinstGate_2(iniHomePos := "FG_TS_Gate_2_InHome",   // "Cylinder_1Out2In"
                iniWorkPos := "FG_TS_Gate_2_InWork",
                configNoReleaseCycle := true,
                actor := "TransportActors".Gate_2,
                signals := #signals,
                manualMovement := #manualMovements,
                workPos => "FG_TS_Gate_2_WorkPos");
END_REGION

REGION Network 3: Reserved
   #instActorReserved1(manualMovement := #manualMovements);   // "Actor_Reserved"
END_REGION

REGION Network 4: Reserved
   #instActorReserved2(manualMovement := #manualMovements);   // "Actor_Reserved"
END_REGION

REGION Network 5: Index01 Y-Lift
   #sinstIndex01_Y_Lift(iniHomePos := "FG_TS_Index01_Y_Lift_InHome",   // "Cylinder_2Out2In"
                        iniWorkPos := "FG_TS_Index01_Y_Lift_InWork",
                        actor := "TransportActors".Index01_Lift,
                        signals := #signals,
                        manualMovement := #manualMovements,
                        homePos => "FG_TS_Index01_Y_Lift_HomePos",
                        workPos => "FG_TS_Index01_Y_Lift_WorkPos");
END_REGION

REGION Network 6: Index01 Y-Stopper
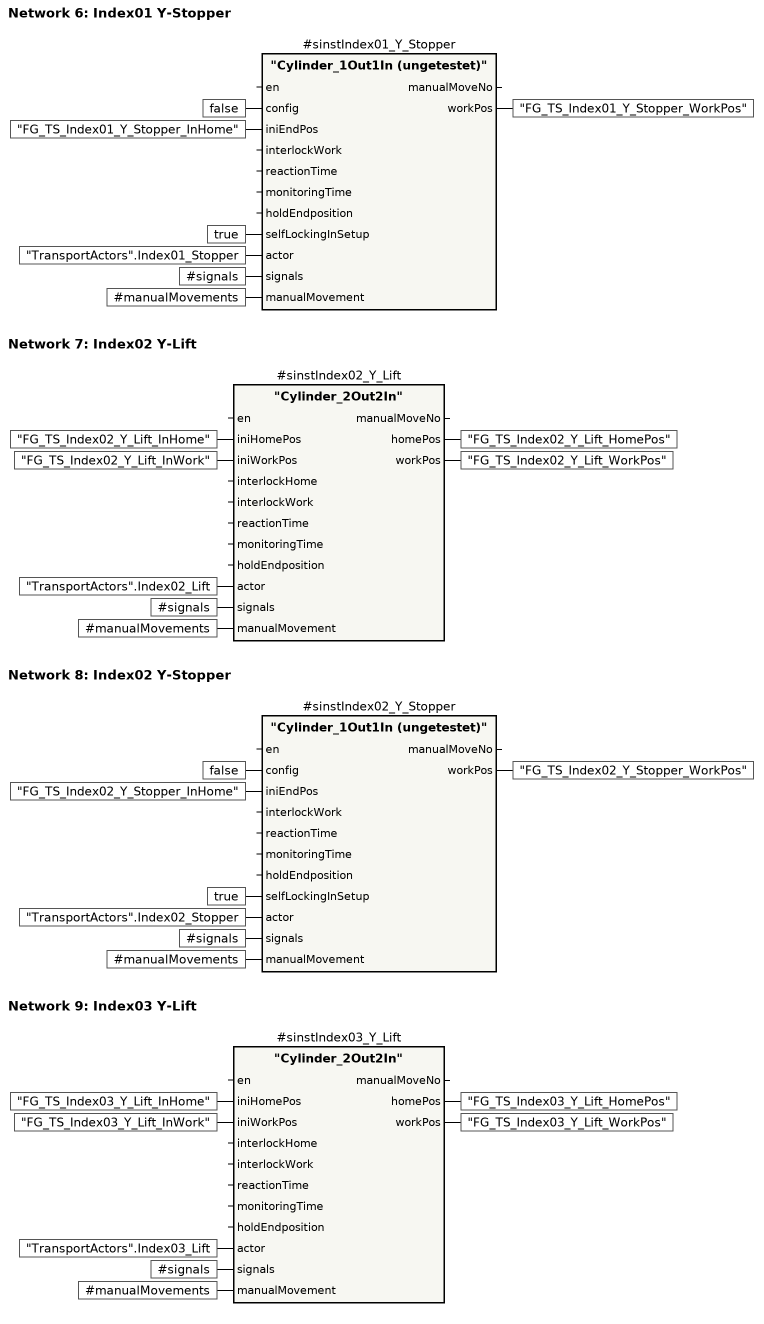
   #sinstIndex01_Y_Stopper(config := false,   // "Cylinder_1Out1In (ungetestet)"
                           iniEndPos := "FG_TS_Index01_Y_Stopper_InHome",
                           selfLockingInSetup := true,
                           actor := "TransportActors".Index01_Stopper,
                           signals := #signals,
                           manualMovement := #manualMovements,
                           workPos => "FG_TS_Index01_Y_Stopper_WorkPos");
END_REGION

REGION Network 7: Index02 Y-Lift
   #sinstIndex02_Y_Lift(iniHomePos := "FG_TS_Index02_Y_Lift_InHome",   // "Cylinder_2Out2In"
                        iniWorkPos := "FG_TS_Index02_Y_Lift_InWork",
                        actor := "TransportActors".Index02_Lift,
                        signals := #signals,
                        manualMovement := #manualMovements,
                        homePos => "FG_TS_Index02_Y_Lift_HomePos",
                        workPos => "FG_TS_Index02_Y_Lift_WorkPos");
END_REGION

REGION Network 8: Index02 Y-Stopper
   #sinstIndex02_Y_Stopper(config := false,   // "Cylinder_1Out1In (ungetestet)"
                           iniEndPos := "FG_TS_Index02_Y_Stopper_InHome",
                           selfLockingInSetup := true,
                           actor := "TransportActors".Index02_Stopper,
                           signals := #signals,
                           manualMovement := #manualMovements,
                           workPos => "FG_TS_Index02_Y_Stopper_WorkPos");
END_REGION

REGION Network 9: Index03 Y-Lift
   #sinstIndex03_Y_Lift(iniHomePos := "FG_TS_Index03_Y_Lift_InHome",   // "Cylinder_2Out2In"
                        iniWorkPos := "FG_TS_Index03_Y_Lift_InWork",
                        actor := "TransportActors".Index03_Lift,
                        signals := #signals,
                        manualMovement := #manualMovements,
                        homePos => "FG_TS_Index03_Y_Lift_HomePos",
                        workPos => "FG_TS_Index03_Y_Lift_WorkPos");
END_REGION

REGION Network 10: Index03 Y-Stopper
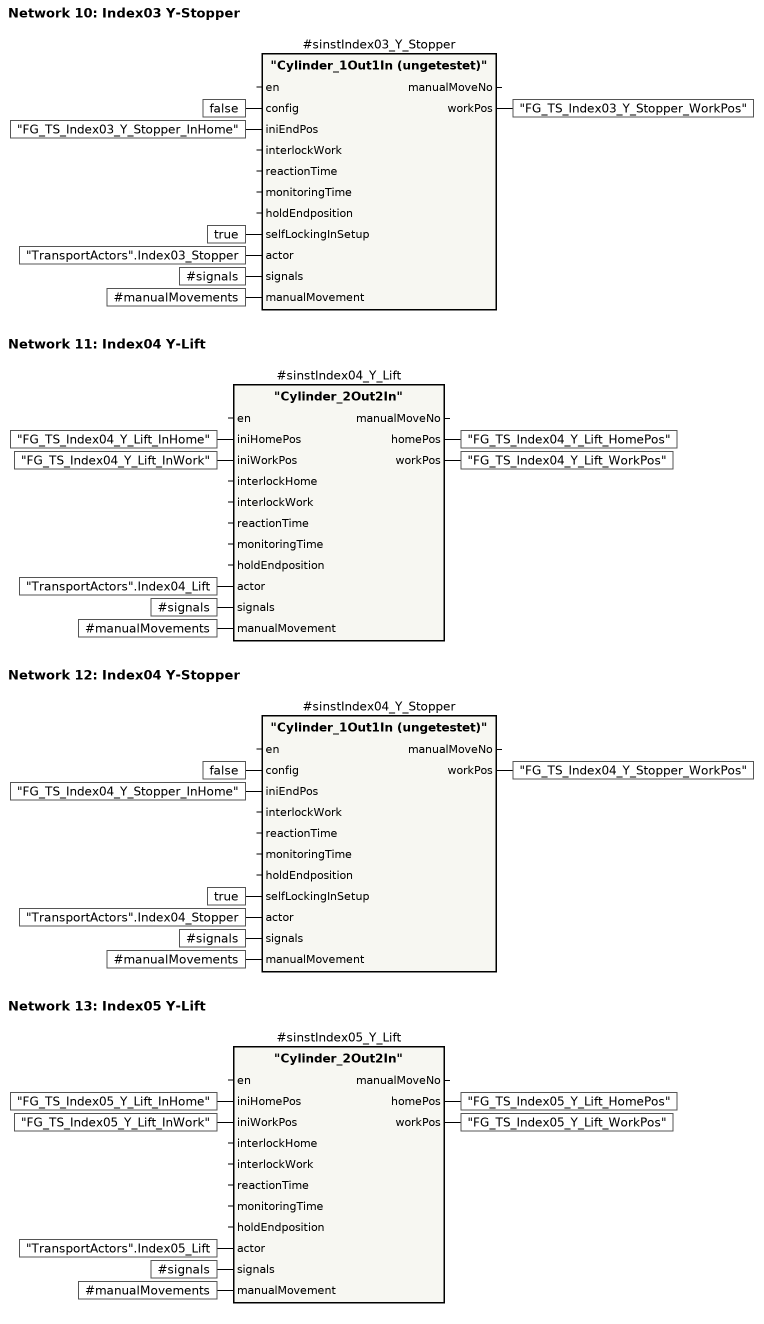
   #sinstIndex03_Y_Stopper(config := false,   // "Cylinder_1Out1In (ungetestet)"
                           iniEndPos := "FG_TS_Index03_Y_Stopper_InHome",
                           selfLockingInSetup := true,
                           actor := "TransportActors".Index03_Stopper,
                           signals := #signals,
                           manualMovement := #manualMovements,
                           workPos => "FG_TS_Index03_Y_Stopper_WorkPos");
END_REGION

REGION Network 11: Index04 Y-Lift
   #sinstIndex04_Y_Lift(iniHomePos := "FG_TS_Index04_Y_Lift_InHome",   // "Cylinder_2Out2In"
                        iniWorkPos := "FG_TS_Index04_Y_Lift_InWork",
                        actor := "TransportActors".Index04_Lift,
                        signals := #signals,
                        manualMovement := #manualMovements,
                        homePos => "FG_TS_Index04_Y_Lift_HomePos",
                        workPos => "FG_TS_Index04_Y_Lift_WorkPos");
END_REGION

REGION Network 12: Index04 Y-Stopper
   #sinstIndex04_Y_Stopper(config := false,   // "Cylinder_1Out1In (ungetestet)"
                           iniEndPos := "FG_TS_Index04_Y_Stopper_InHome",
                           selfLockingInSetup := true,
                           actor := "TransportActors".Index04_Stopper,
                           signals := #signals,
                           manualMovement := #manualMovements,
                           workPos => "FG_TS_Index04_Y_Stopper_WorkPos");
END_REGION

REGION Network 13: Index05 Y-Lift
   #sinstIndex05_Y_Lift(iniHomePos := "FG_TS_Index05_Y_Lift_InHome",   // "Cylinder_2Out2In"
                        iniWorkPos := "FG_TS_Index05_Y_Lift_InWork",
                        actor := "TransportActors".Index05_Lift,
                        signals := #signals,
                        manualMovement := #manualMovements,
                        homePos => "FG_TS_Index05_Y_Lift_HomePos",
                        workPos => "FG_TS_Index05_Y_Lift_WorkPos");
END_REGION

REGION Network 14: Index05 Y-Stopper
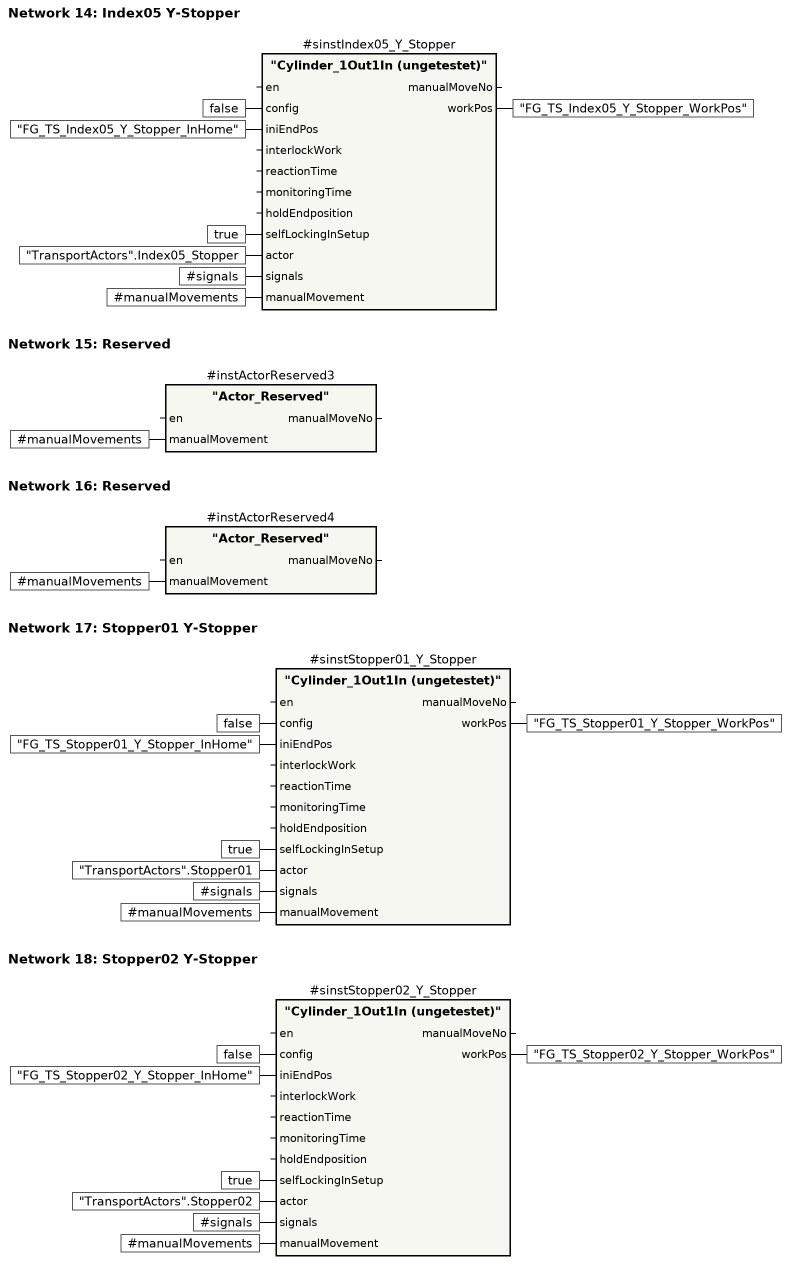
   #sinstIndex05_Y_Stopper(config := false,   // "Cylinder_1Out1In (ungetestet)"
                           iniEndPos := "FG_TS_Index05_Y_Stopper_InHome",
                           selfLockingInSetup := true,
                           actor := "TransportActors".Index05_Stopper,
                           signals := #signals,
                           manualMovement := #manualMovements,
                           workPos => "FG_TS_Index05_Y_Stopper_WorkPos");
END_REGION

REGION Network 15: Reserved
   #instActorReserved3(manualMovement := #manualMovements);   // "Actor_Reserved"
END_REGION

REGION Network 16: Reserved
   #instActorReserved4(manualMovement := #manualMovements);   // "Actor_Reserved"
END_REGION

REGION Network 17: Stopper01 Y-Stopper
   #sinstStopper01_Y_Stopper(config := false,   // "Cylinder_1Out1In (ungetestet)"
                           iniEndPos := "FG_TS_Stopper01_Y_Stopper_InHome",
                           selfLockingInSetup := true,
                           actor := "TransportActors".Stopper01,
                           signals := #signals,
                           manualMovement := #manualMovements,
                           workPos => "FG_TS_Stopper01_Y_Stopper_WorkPos");
END_REGION

REGION Network 18: Stopper02 Y-Stopper
   #sinstStopper02_Y_Stopper(config := false,   // "Cylinder_1Out1In (ungetestet)"
                           iniEndPos := "FG_TS_Stopper02_Y_Stopper_InHome",
                           selfLockingInSetup := true,
                           actor := "TransportActors".Stopper02,
                           signals := #signals,
                           manualMovement := #manualMovements,
                           workPos => "FG_TS_Stopper02_Y_Stopper_WorkPos");
END_REGION

REGION Network 19: Stopper03 Y-Stopper
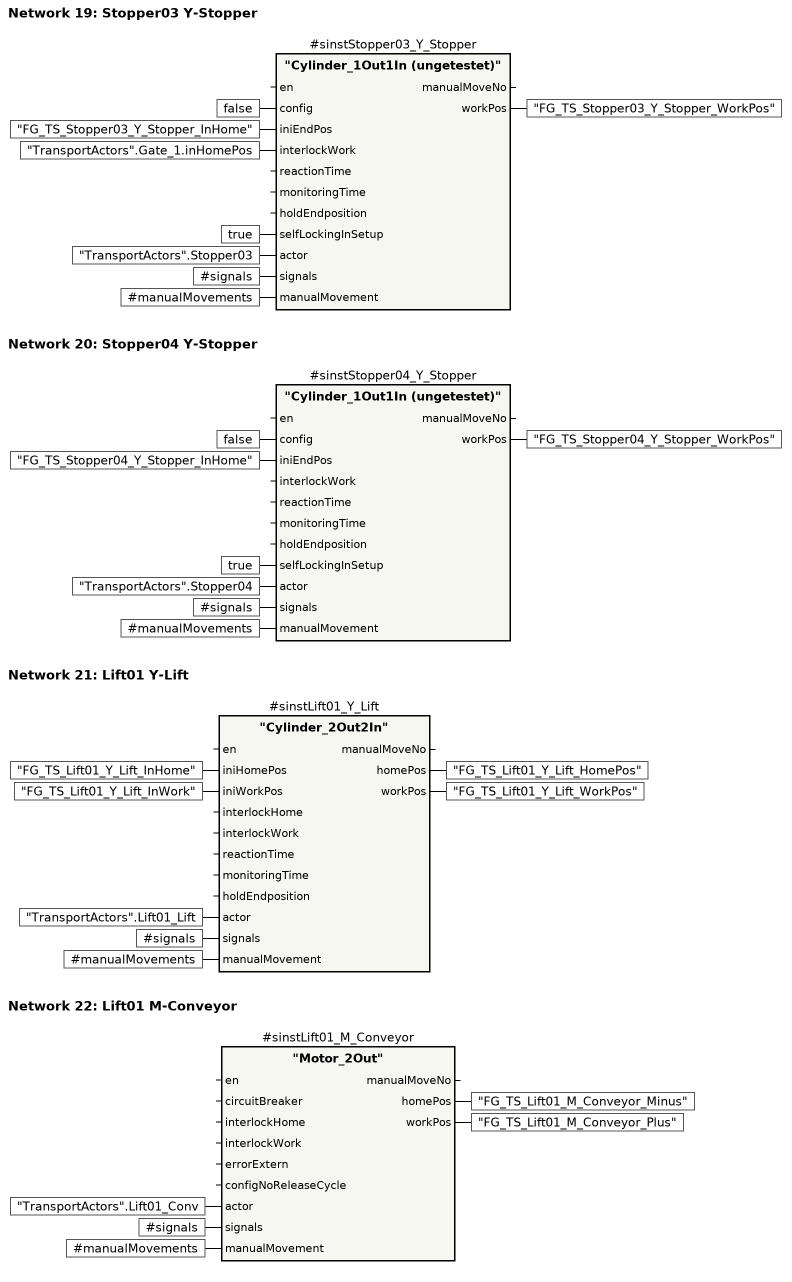
   #sinstStopper03_Y_Stopper(config := false,   // "Cylinder_1Out1In (ungetestet)"
                           iniEndPos := "FG_TS_Stopper03_Y_Stopper_InHome",
                           interlockWork := "TransportActors".Gate_1.inHomePos,
                           selfLockingInSetup := true,
                           actor := "TransportActors".Stopper03,
                           signals := #signals,
                           manualMovement := #manualMovements,
                           workPos => "FG_TS_Stopper03_Y_Stopper_WorkPos");
END_REGION

REGION Network 20: Stopper04 Y-Stopper
   #sinstStopper04_Y_Stopper(config := false,   // "Cylinder_1Out1In (ungetestet)"
                           iniEndPos := "FG_TS_Stopper04_Y_Stopper_InHome",
                           selfLockingInSetup := true,
                           actor := "TransportActors".Stopper04,
                           signals := #signals,
                           manualMovement := #manualMovements,
                           workPos => "FG_TS_Stopper04_Y_Stopper_WorkPos");
END_REGION

REGION Network 21: Lift01 Y-Lift
   #sinstLift01_Y_Lift(iniHomePos := "FG_TS_Lift01_Y_Lift_InHome",   // "Cylinder_2Out2In"
                       iniWorkPos := "FG_TS_Lift01_Y_Lift_InWork",
                       actor := "TransportActors".Lift01_Lift,
                       signals := #signals,
                       manualMovement := #manualMovements,
                       homePos => "FG_TS_Lift01_Y_Lift_HomePos",
                       workPos => "FG_TS_Lift01_Y_Lift_WorkPos");
END_REGION

REGION Network 22: Lift01 M-Conveyor
   #sinstLift01_M_Conveyor(actor := "TransportActors".Lift01_Conv,   // "Motor_2Out"
                           signals := #signals,
                           manualMovement := #manualMovements,
                           homePos => "FG_TS_Lift01_M_Conveyor_Minus",
                           workPos => "FG_TS_Lift01_M_Conveyor_Plus");
END_REGION

REGION Network 23: Lift02 Y-Lift
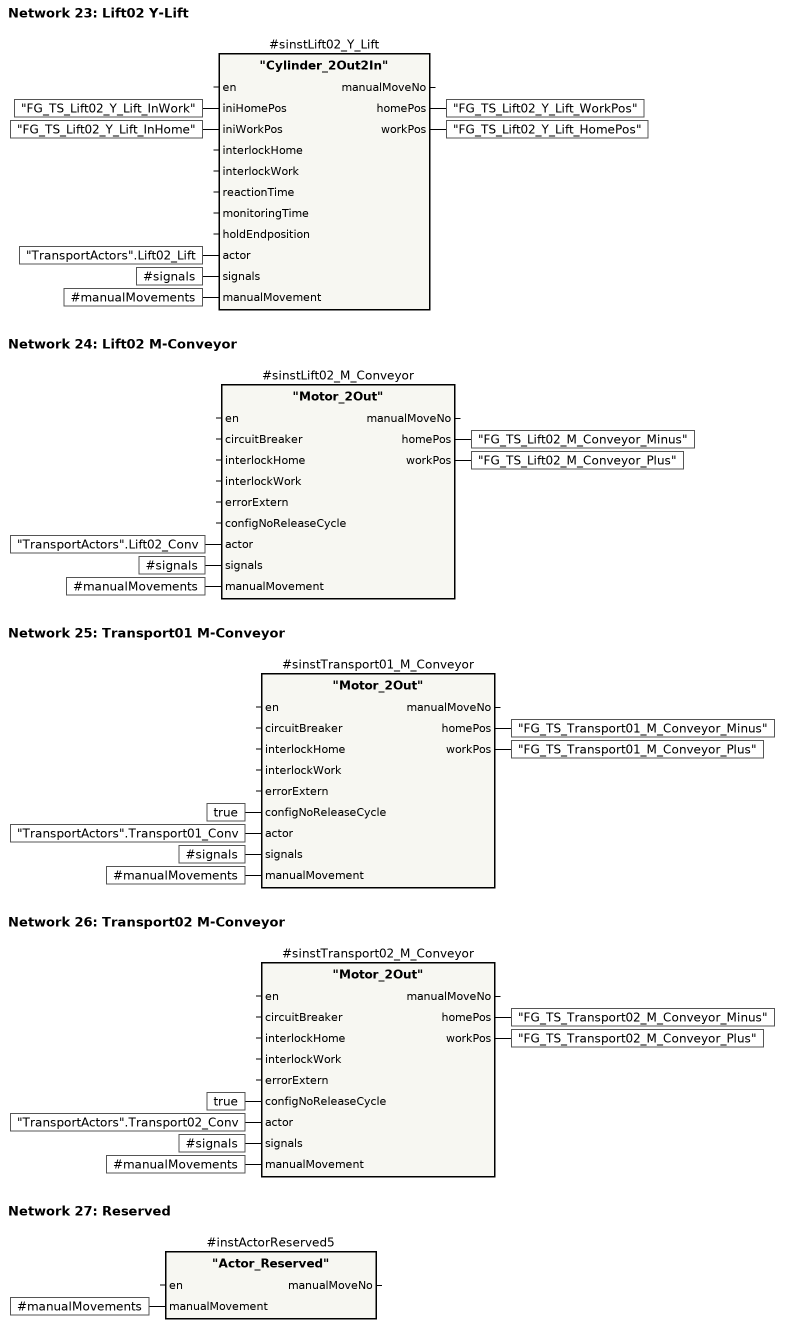
   #sinstLift02_Y_Lift(iniHomePos := "FG_TS_Lift02_Y_Lift_InWork",   // "Cylinder_2Out2In"
                       iniWorkPos := "FG_TS_Lift02_Y_Lift_InHome",
                       actor := "TransportActors".Lift02_Lift,
                       signals := #signals,
                       manualMovement := #manualMovements,
                       homePos => "FG_TS_Lift02_Y_Lift_WorkPos",
                       workPos => "FG_TS_Lift02_Y_Lift_HomePos");
END_REGION

REGION Network 24: Lift02 M-Conveyor
   #sinstLift02_M_Conveyor(actor := "TransportActors".Lift02_Conv,   // "Motor_2Out"
                           signals := #signals,
                           manualMovement := #manualMovements,
                           homePos => "FG_TS_Lift02_M_Conveyor_Minus",
                           workPos => "FG_TS_Lift02_M_Conveyor_Plus");
END_REGION

REGION Network 25: Transport01 M-Conveyor
   #sinstTransport01_M_Conveyor(configNoReleaseCycle := true,   // "Motor_2Out"
                           actor := "TransportActors".Transport01_Conv,
                           signals := #signals,
                           manualMovement := #manualMovements,
                           homePos => "FG_TS_Transport01_M_Conveyor_Minus",
                           workPos => "FG_TS_Transport01_M_Conveyor_Plus");
END_REGION

REGION Network 26: Transport02 M-Conveyor
   #sinstTransport02_M_Conveyor(configNoReleaseCycle := true,   // "Motor_2Out"
                           actor := "TransportActors".Transport02_Conv,
                           signals := #signals,
                           manualMovement := #manualMovements,
                           homePos => "FG_TS_Transport02_M_Conveyor_Minus",
                           workPos => "FG_TS_Transport02_M_Conveyor_Plus");
END_REGION

REGION Network 27: Reserved
   #instActorReserved5(manualMovement := #manualMovements);   // "Actor_Reserved"
END_REGION

REGION Network 28: Reserved
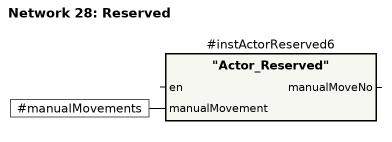
   #instActorReserved6(manualMovement := #manualMovements);   // "Actor_Reserved"
END_REGION
END_FUNCTION_BLOCK

// folder: 2. Machine/10_FG_Transport/Stepsequences

FUNCTION_BLOCK "Sq_Process_IndexingUnit01"   // FB2111, GRAPH_PLUS
{ S7_Optimized_Access := 'TRUE' }
VERSION : 0.1
   VAR_INPUT
      OFF_SQ : Bool := false;   // Kette ausschalten
      INIT_SQ : Bool := false;   // Kette in Initialzustand versetzen
      ACK_EF : Bool := false;   // Alle Fehler und Störungen quittieren
      S_PREV : Bool := false;   // Vorherigen Schritt am Parameter S_NO ausgeben
      S_NEXT : Bool := false;   // Nächsten Schritt am Parameter S_NO anzeigen
      SW_AUTO : Bool := false;   // Automatischer Betrieb
      SW_TAP : Bool := false;   // Halbautomatisch/Weiterschalten mit Transition
      SW_TOP : Bool := false;   // Halbautomatisch/Ignoriere Transition
      SW_MAN : Bool := false;   // Handbetrieb
      S_SEL : Int := 0;   // Schritt auswählen, der an S_NO ausgegeben werden soll
      S_ON : Bool := false;   // Schritt aktivieren, der an Parameter S_NO anliegt
      S_OFF : Bool := false;   // Schritt deaktivieren, der an Parameter S_NO anliegt
      T_PUSH : Bool := false;   // Schaltfreigabe für Transition im halbautomatischen Betrieb
      ixStart : Bool := true;   // Startfreigabe
      ixCarrierPresent : Bool;   // WT auf dem Indexer vorhanden
      ixCheckTargetReached : Bool := false;   // 0 = Keine Sensor-Zielüberwachung nach Lift vorhanden
      ixTargetReached : Bool := false;   // WT-Sensor des nächsten Ziels
      ixReleaseHoming : Bool;   // Freigabe Grundstellungsfahrt
      ixReleaseTransfer : Bool := true;   // Freigabe der nächsten Position um WT weiterzutakten
      itCarrierReactionDelay : Time := T#350ms;   // Verzögerungszeit für die WT-Erkennung
      itMaxRuntime : Time := t#10s;   // Maximale Laufzeit für diesen Prozess
   END_VAR
   VAR_OUTPUT
      S_NO : Int := 0;   // Schrittnummer
      S_MORE : Bool := false;   // Weitere Schritte sind vorhanden und können in S_NO angezeigt werden.
      S_ACTIVE : Bool := false;   // Schritt, der an Parameter S_NO angezeigt wird, ist aktiv
      ERR_FLT : Bool := false;   // Sammelfehler Interlock oder Supervision
      AUTO_ON : Bool := false;   // Automatischer Betrieb eingeschaltet
      TAP_ON : Bool := false;   // Halbautomatischer Betrieb/Schritt mit Transition eingeschaltet
      TOP_ON : Bool := false;   // Halbautomatischer Betrieb/Ignoriere Transition eingeschaltet
      MAN_ON : Bool := false;   // Handbetrieb eingeschaltet
      qxIsActive : Bool;   // Schrittkette läuft
      qxIsInHome : Bool;   // steht in Grundstellung
      qxCarrierIsDone : Bool;   // WT-Träger ist fertig bearbeitet worden
   END_VAR
   VAR_IN_OUT
      signals : "typeStationSignals";   // Stationssteuersignale
      sq : "typeStepSequence";   // Schrittkettensteuersignale
      cylinder_lift : "typeActor_2Out2In";   // Aktor des Heber
      cylinder_stopper : "typeActor_1Out1In";   // Aktor für den Stopper
      releaseWorkStep : Bool;   // Freigabe für den externen Arbeitsschritt (muss extern zurückgesetzt werden)
   END_VAR
   VAR
      sstReleaseCycle : Struct
         ErrorAck : Bool;
         No_LastCycle : Int;
         T : Time;   // Aktive Zeit des ReleaseCycle
         Tck : Time;
         TckPrev : Time;
      END_STRUCT;
      sinstCarrierOnIndexer : TON_TIME;
      sinstCarrierLeftIndexer : TON_TIME;
      sxTrigReleaseWorkStep : Bool;
      HMI_INFO : Array[0..8] of UInt;
      IF_PAR : G7_IfParPlus_V6;
      RT_DATA : G7_RTDataPlus_V6;   // Interner Datenbereich
      Automatikablauf : G7_TransitionPlus_V6;   // Transitionsstruktur
      Freigabe : G7_TransitionPlus_V6;   // Transitionsstruktur
      Trans3 : G7_TransitionPlus_V6;   // Transitionsstruktur
      Fertig : G7_TransitionPlus_V6;   // Transitionsstruktur / Transition structure
      Grundstellungsfahrt : G7_TransitionPlus_V6;   // Transitionsstruktur
      GST_Aktiv : G7_TransitionPlus_V6;   // Transitionsstruktur
      GST_Beendet : G7_TransitionPlus_V6;   // Transitionsstruktur
      Beendet : G7_TransitionPlus_V6;   // Transitionsstruktur
      TargetIsReached : G7_TransitionPlus_V6;   // Transitionsstruktur / Transition structure
      "Lift steht in Grundstellung_1" : G7_TransitionPlus_V6;   // Transitionsstruktur / Transition structure
      "Lift steht in Arbeitsstellung_1" : G7_TransitionPlus_V6;   // Transitionsstruktur / Transition structure
      "Lift steht in Arbeitsstellung_2" : G7_TransitionPlus_V6;   // Transitionsstruktur / Transition structure
      "WT hat Stopper verlassen" : G7_TransitionPlus_V6;   // Transitionsstruktur / Transition structure
      CarrierIsNotDone : G7_TransitionPlus_V6;   // Transitionsstruktur / Transition structure
      CarrierIsDone : G7_TransitionPlus_V6;   // Transitionsstruktur / Transition structure
      WorkstepIsReleased : G7_TransitionPlus_V6;   // Transitionsstruktur / Transition structure
      GS_ReleaseReseted : G7_TransitionPlus_V6;   // Transitionsstruktur / Transition structure
      GS_NoCarrier : G7_TransitionPlus_V6;   // Transitionsstruktur / Transition structure
      GS_CarrierOnIndexer : G7_TransitionPlus_V6;   // Transitionsstruktur / Transition structure
      JogT4 : G7_TransitionPlus_V6;   // Transitionsstruktur / Transition structure
      JogT1 : G7_TransitionPlus_V6;   // Transitionsstruktur / Transition structure
      GatesClosed : G7_TransitionPlus_V6;   // Transitionsstruktur / Transition structure
      GatesOpened : G7_TransitionPlus_V6;   // Transitionsstruktur / Transition structure
      JogT3 : G7_TransitionPlus_V6;   // Transitionsstruktur / Transition structure
      GS_GatesOpened : G7_TransitionPlus_V6;   // Transitionsstruktur / Transition structure
      GS_Reseted : G7_TransitionPlus_V6;   // Transitionsstruktur / Transition structure
      Initialschritt : G7_StepPlus_V6;   // Schrittstruktur
      Grundstellung : G7_StepPlus_V6;   // Schrittstruktur
      SK_läuft : G7_StepPlus_V6;   // Schrittstruktur
      Fertigmeldung : G7_StepPlus_V6;   // Schrittstruktur / Step structure
      "Start Grundstellungsfahrt" : G7_StepPlus_V6;   // Schrittstruktur
      "Fertig Grundstellungsfahrt" : G7_StepPlus_V6;   // Schrittstruktur
      Ende : G7_StepPlus_V6;   // Schrittstruktur
      WaitForTarget : G7_StepPlus_V6;   // Schrittstruktur / Step structure
      GS_CylHome : G7_StepPlus_V6;   // Schrittstruktur / Step structure
      IndexerWorkPos : G7_StepPlus_V6;   // Schrittstruktur / Step structure
      IndexerHomePos : G7_StepPlus_V6;   // Schrittstruktur / Step structure
      OpenStopper : G7_StepPlus_V6;   // Schrittstruktur / Step structure
      Decision : G7_StepPlus_V6;   // Schrittstruktur / Step structure
      Release : G7_StepPlus_V6;   // Schrittstruktur / Step structure
      GS_ResetRelease : G7_StepPlus_V6;   // Schrittstruktur / Step structure
      GS_CheckCarrier : G7_StepPlus_V6;   // Schrittstruktur / Step structure
      GS_ResetCarrierIsDone : G7_StepPlus_V6;   // Schrittstruktur / Step structure
      JogS4 : G7_StepPlus_V6;   // Schrittstruktur / Step structure
      JogS1 : G7_StepPlus_V6;   // Schrittstruktur / Step structure
      CloseGates : G7_StepPlus_V6;   // Schrittstruktur / Step structure
      OpenGates : G7_StepPlus_V6;   // Schrittstruktur / Step structure
      JogS3 : G7_StepPlus_V6;   // Schrittstruktur / Step structure
      GS_OpenGates : G7_StepPlus_V6;   // Schrittstruktur / Step structure
      SINI : Array[0..1] of USInt;
      LSTT : Array[0..25] of USInt;
      ATAJ : Array[0..25] of USInt;
      ATAB : Array[0..25] of USInt;
      PSTT : Array[0..25] of USInt;
      NSTT : Array[0..25] of USInt;
      ASSJ : Array[0..22] of USInt;
      ASSB : Array[0..22] of USInt;
      PTTS : Array[0..22] of USInt;
      NTTS : Array[0..22] of USInt;
      SW_SQTS : Array[0..22] of USInt;
      SWITCH : Array[0..7] of USInt;
      TVX : Array[0..7] of USInt;
      TTX : Array[0..7] of USInt;
      TSX : Array[0..1] of USInt;
      S00X : Array[0..1] of USInt;
      SOFFX : Array[0..1] of USInt;
      SONX : Array[0..1] of USInt;
      SAX : Array[0..1] of USInt;
      SERRX : Array[0..23] of USInt;
      SMX : Array[0..23] of USInt;
      S0X : Array[0..23] of USInt;
      S1X : Array[0..23] of USInt;
      IL_ALARM_INST : Diag_Alarm;
      SUP_ALARM_INST : Diag_Alarm;
      STEP_TIME_ALARM_INST : Diag_Alarm;
      IEC_TIMER_INST : IEC_TIMER;
      TRANSACTION_FLAG : Bool := false;
   END_VAR
   VAR_TEMP
      txStartCondition : Bool;
      tdTckDiff : DInt;
      txStartNewCarrier : Bool;
      txCarrierIsDone : Bool;
   END_VAR
   VAR_TEMP   // added for the SCL form of the ladder/FBD networks
      _w1 : Bool;
      _w2 : Bool;
   END_VAR
   // SINI[0] := 2;
   // LSTT[0] := 255;
   // LSTT[1] := 255;
   // LSTT[2] := 255;
   // LSTT[3] := 255;
   // LSTT[4] := 255;
   // LSTT[5] := 255;
   // LSTT[6] := 255;
   // LSTT[7] := 1;
   // ATAJ[1] := 1;
   // ATAJ[2] := 2;
   // ATAJ[3] := 6;
   // ATAJ[4] := 4;
   // ATAJ[5] := 5;
   // ATAJ[6] := 15;
   // ATAJ[7] := 7;
   // ATAB[0] := 4;
   // ATAB[1] := 1;
   // ATAB[2] := 2;
   // ATAB[3] := 3;
   // ATAB[5] := 5;
   // ATAB[6] := 6;
   // ATAB[7] := 7;
   // PSTT[1] := 1;
   // PSTT[2] := 2;
   // PSTT[3] := 3;
   // PSTT[5] := 4;
   // PSTT[6] := 5;
   // PSTT[7] := 6;
   // NSTT[0] := 1;
   // NSTT[1] := 2;
   // NSTT[2] := 12;
   // NSTT[3] := 6;
   // NSTT[4] := 4;
   // NSTT[5] := 14;
   // NSTT[6] := 6;
   // NSTT[7] := 1;
   // ASSJ[1] := 1;
   // ASSJ[2] := 2;
   // ASSJ[3] := 3;
   // ASSJ[4] := 4;
   // ASSJ[5] := 5;
   // ASSJ[6] := 6;
   // ASSB[1] := 1;
   // ASSB[2] := 2;
   // ASSB[3] := 3;
   // ASSB[4] := 4;
   // ASSB[5] := 5;
   // ASSB[6] := 6;
   // PTTS[0] := 255;
   // PTTS[2] := 1;
   // PTTS[3] := 8;
   // PTTS[4] := 4;
   // PTTS[5] := 24;
   // PTTS[6] := 15;
   // NTTS[1] := 1;
   // NTTS[2] := 2;
   // NTTS[3] := 3;
   // NTTS[4] := 5;
   // NTTS[5] := 6;
   // NTTS[6] := 7;
   // SW_SQTS[1] := 1;
   // SW_SQTS[2] := 1;
   // SW_SQTS[3] := 2;
   // SW_SQTS[4] := 3;
   // SW_SQTS[5] := 4;
   // SW_SQTS[6] := 5;
   // TVX[0] := 16#1;
   // TTX[0] := 16#1;
   // TSX[0] := 16#1;
   // S00X[0] := 16#1;
   // SOFFX[0] := 16#1;
   // SONX[0] := 16#1;
   // SAX[0] := 16#1;
   // SERRX[0] := 16#1;
   // SMX[0] := 16#1;
   // S0X[0] := 16#1;
   // S1X[0] := 16#1;
   // LSTT[8] := 255;
   // ATAJ[8] := 8;
   // ATAB[8] := 8;
   // PSTT[8] := 7;
   // NSTT[8] := 3;
   // ASSJ[7] := 7;
   // ASSB[7] := 7;
   // PTTS[7] := 12;
   // NTTS[7] := 8;
   // SW_SQTS[7] := 2;
   // LSTT[9] := 255;
   // LSTT[10] := 255;
   // LSTT[11] := 255;
   // ATAJ[9] := 9;
   // ATAJ[10] := 10;
   // ATAJ[11] := 11;
   // ATAB[9] := 9;
   // ATAB[10] := 10;
   // ATAB[11] := 11;
   // PSTT[9] := 8;
   // PSTT[10] := 9;
   // PSTT[11] := 10;
   // NSTT[9] := 22;
   // NSTT[10] := 18;
   // NSTT[11] := 17;
   // ASSJ[8] := 8;
   // ASSJ[9] := 9;
   // ASSJ[10] := 10;
   // ASSB[8] := 8;
   // ASSB[9] := 9;
   // ASSB[10] := 10;
   // PTTS[8] := 25;
   // PTTS[9] := 13;
   // PTTS[10] := 23;
   // NTTS[8] := 9;
   // NTTS[9] := 10;
   // NTTS[10] := 11;
   // SW_SQTS[8] := 4;
   // SW_SQTS[9] := 6;
   // SW_SQTS[10] := 2;
   // LSTT[12] := 255;
   // LSTT[13] := 255;
   // ATAJ[12] := 12;
   // ATAJ[13] := 13;
   // ATAB[12] := 12;
   // ATAB[13] := 14;
   // PSTT[12] := 11;
   // PSTT[13] := 12;
   // NSTT[12] := 7;
   // NSTT[13] := 9;
   // ASSJ[11] := 11;
   // ASSJ[12] := 12;
   // ASSB[11] := 11;
   // ASSB[12] := 12;
   // PTTS[11] := 19;
   // PTTS[12] := 2;
   // NTTS[11] := 12;
   // NTTS[12] := 13;
   // SW_SQTS[11] := 2;
   // SW_SQTS[12] := 1;
   // LSTT[14] := 255;
   // LSTT[15] := 255;
   // ATAJ[14] := 14;
   // ATAJ[15] := 3;
   // ATAB[14] := 13;
   // ATAB[15] := 15;
   // PSTT[14] := 12;
   // PSTT[15] := 13;
   // NSTT[14] := 20;
   // NSTT[15] := 6;
   // ASSJ[13] := 13;
   // ASSJ[14] := 14;
   // ASSB[13] := 13;
   // ASSB[14] := 14;
   // PTTS[13] := 21;
   // PTTS[14] := 5;
   // NTTS[13] := 15;
   // NTTS[14] := 16;
   // SW_SQTS[13] := 6;
   // SW_SQTS[14] := 3;
   // LSTT[16] := 255;
   // ATAJ[16] := 16;
   // ATAB[16] := 16;
   // PSTT[16] := 14;
   // NSTT[16] := 15;
   // LSTT[17] := 255;
   // LSTT[18] := 255;
   // ATAJ[17] := 17;
   // ATAJ[18] := 25;
   // ATAB[17] := 18;
   // ATAB[18] := 17;
   // PSTT[17] := 15;
   // PSTT[18] := 15;
   // NSTT[17] := 16;
   // NSTT[18] := 8;
   // ASSJ[15] := 15;
   // ASSB[15] := 15;
   // PTTS[15] := 16;
   // NTTS[15] := 17;
   // SW_SQTS[15] := 3;
   // LSTT[19] := 255;
   // ATAJ[19] := 19;
   // ATAB[19] := 19;
   // PSTT[19] := 17;
   // NSTT[19] := 11;
   // ASSJ[16] := 16;
   // ASSB[16] := 16;
   // PTTS[16] := 17;
   // NTTS[16] := 25;
   // SW_SQTS[16] := 7;
   // LSTT[20] := 255;
   // LSTT[21] := 255;
   // LSTT[22] := 255;
   // ATAJ[20] := 20;
   // ATAJ[21] := 21;
   // ATAJ[22] := 22;
   // ATAB[20] := 20;
   // ATAB[21] := 21;
   // ATAB[22] := 22;
   // PSTT[20] := 18;
   // PSTT[21] := 19;
   // PSTT[22] := 20;
   // NSTT[20] := 19;
   // NSTT[21] := 13;
   // NSTT[22] := 21;
   // ASSJ[17] := 17;
   // ASSJ[18] := 18;
   // ASSJ[19] := 19;
   // ASSJ[20] := 20;
   // ASSB[17] := 17;
   // ASSB[18] := 18;
   // ASSB[19] := 19;
   // ASSB[20] := 20;
   // PTTS[17] := 11;
   // PTTS[18] := 10;
   // PTTS[19] := 20;
   // PTTS[20] := 14;
   // NTTS[17] := 19;
   // NTTS[18] := 20;
   // NTTS[19] := 21;
   // NTTS[20] := 22;
   // SW_SQTS[17] := 2;
   // SW_SQTS[18] := 6;
   // SW_SQTS[19] := 6;
   // SW_SQTS[20] := 2;
   // LSTT[23] := 255;
   // LSTT[24] := 255;
   // LSTT[25] := 255;
   // ATAJ[23] := 23;
   // ATAJ[24] := 24;
   // ATAJ[25] := 18;
   // ATAB[23] := 23;
   // ATAB[24] := 24;
   // ATAB[25] := 25;
   // PSTT[23] := 21;
   // PSTT[24] := 22;
   // PSTT[25] := 16;
   // NSTT[23] := 10;
   // NSTT[24] := 5;
   // NSTT[25] := 8;
   // ASSJ[21] := 21;
   // ASSJ[22] := 22;
   // ASSB[21] := 21;
   // ASSB[22] := 22;
   // PTTS[21] := 22;
   // PTTS[22] := 9;
   // NTTS[21] := 23;
   // NTTS[22] := 24;
   // SW_SQTS[21] := 2;
   // SW_SQTS[22] := 4;
BEGIN
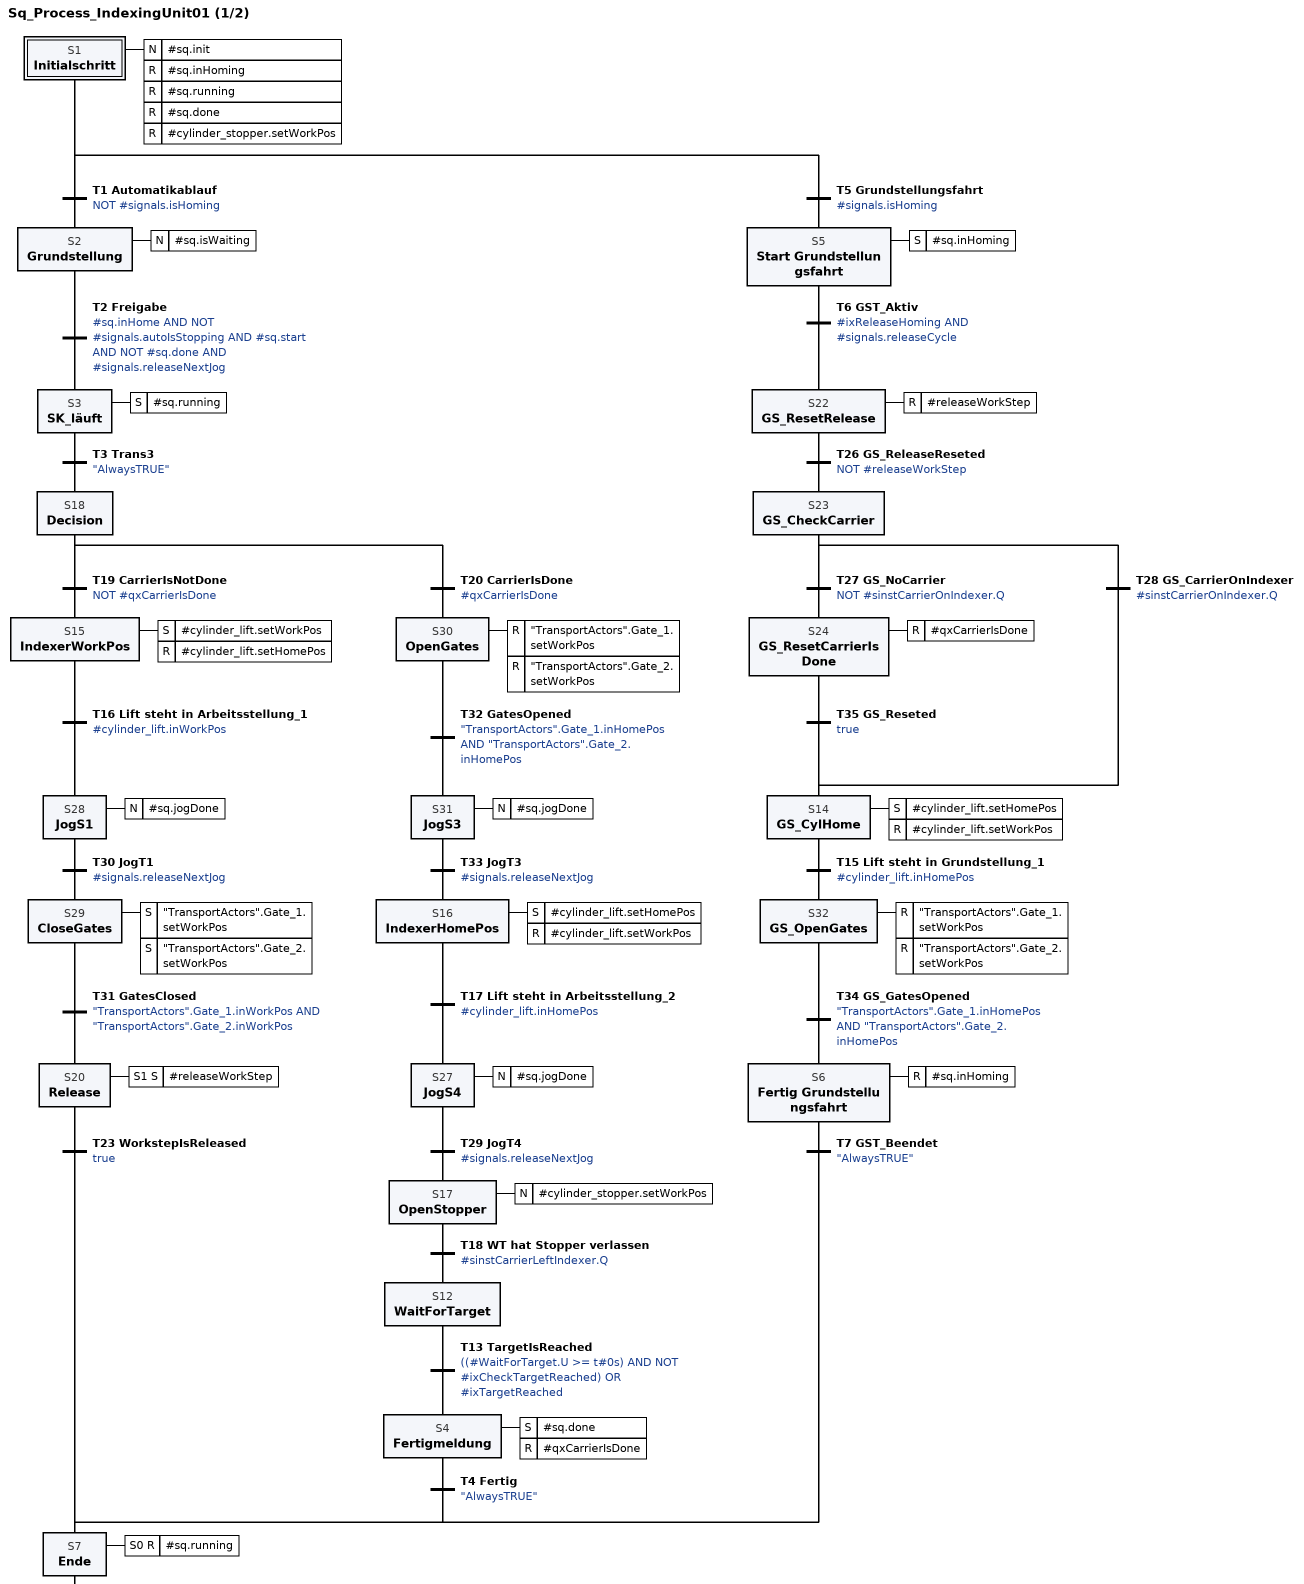
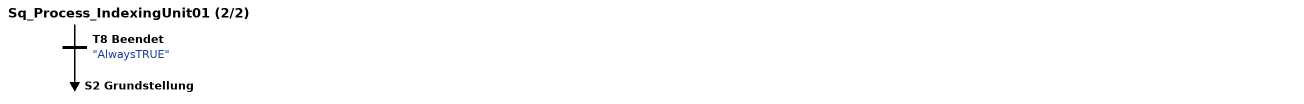
   // permanent pre-instructions
   NETWORK 1
   TITLE = Schrittkette verfügbar
      #sq.exists := true;
   NETWORK 2
   TITLE = WT auf dem Indexer
      #sinstCarrierOnIndexer(IN := #ixCarrierPresent, PT := #itCarrierReactionDelay);   // TON
   NETWORK 3
   TITLE = WT hat den Indexer verlassen
      #sinstCarrierLeftIndexer(IN := NOT #ixCarrierPresent, PT := #itCarrierReactionDelay);   // TON
   NETWORK 4
   TITLE = Schrittkette in Grundstellung (Erweitern)
      #sq.inHome := ((#cylinder_lift.inHomePos AND "TransportActors".Gate_1.inHomePos AND "TransportActors".Gate_2.inHomePos AND NOT #releaseWorkStep) OR (#cylinder_lift.inWorkPos AND "TransportActors".Gate_1.inWorkPos AND "TransportActors".Gate_2.inWorkPos)) AND #Grundstellung.X AND #cylinder_stopper.inHomePos;
   NETWORK 5
   TITLE = Startbedingung (Erweitern)
      #txStartNewCarrier := #ixStart AND #sinstCarrierOnIndexer.Q AND NOT #releaseWorkStep AND NOT #qxCarrierIsDone;
      #txCarrierIsDone := (NOT #ixTargetReached OR NOT #ixCheckTargetReached) AND #ixReleaseTransfer AND #qxCarrierIsDone AND NOT #releaseWorkStep;
      #txStartCondition := #txStartNewCarrier OR #txCarrierIsDone;
   NETWORK 6
   TITLE = Schrittkette starten
      #sq.start := #sq.inHome AND NOT #sq.running AND #signals.releaseCycle AND NOT #signals.isHoming AND #txStartCondition;
      IF #sq.start THEN #sq.done := FALSE; END_IF;
   NETWORK 7
   TITLE = ReleaseCycle Timer
      // ENO of a box is taken as its EN; it also drops when the box reports an error
      #_w1 := #ERR_FLT AND #ACK_EF;
      #_w2 := #_w1 AND NOT #sstReleaseCycle.ErrorAck;   // rising edge
      #sstReleaseCycle.ErrorAck := #_w1;
      IF (#S_NO <> #sstReleaseCycle.No_LastCycle) OR #_w2 THEN
          #sstReleaseCycle.T := T#0MS;
          #sstReleaseCycle.TckPrev := #sstReleaseCycle.Tck;
          #sstReleaseCycle.No_LastCycle := #S_NO;
      END_IF;
      #sstReleaseCycle.Tck := TIME_TCK();
      #tdTckDiff := #sstReleaseCycle.Tck - #sstReleaseCycle.TckPrev;
      #sstReleaseCycle.TckPrev := #sstReleaseCycle.Tck;
      IF (0 <= #tdTckDiff) AND (#tdTckDiff <= 1000) AND #signals.releaseCycle THEN
          #sstReleaseCycle.T := #sstReleaseCycle.T + #tdTckDiff;
      END_IF;

   // sequencer 1
   INITIAL_STEP Initialschritt:   // S1, max time T#10S, warning time T#7S
              N    #sq.init
              R    #sq.inHoming
              R    #sq.running
              R    #sq.done
              R    #cylinder_stopper.setWorkPos
   END_STEP
   TRANSITION Automatikablauf FROM Initialschritt TO Grundstellung   // T1
      := NOT #signals.isHoming;
   END_TRANSITION
   TRANSITION Grundstellungsfahrt FROM Initialschritt TO "Start Grundstellungsfahrt"   // T5
      := #signals.isHoming;
   END_TRANSITION
   STEP Grundstellung:   // S2, max time T#10S, warning time T#7S
              N    #sq.isWaiting
   END_STEP
   TRANSITION Freigabe FROM Grundstellung TO SK_läuft   // T2
      := #sq.inHome AND NOT #signals.autoIsStopping AND #sq.start AND NOT #sq.done AND #signals.releaseNextJog;
   END_TRANSITION
   STEP SK_läuft:   // S3, max time T#10S, warning time T#7S
              S    #sq.running
   END_STEP
   TRANSITION Trans3 FROM SK_läuft TO Decision   // T3
      := "AlwaysTRUE";
   END_TRANSITION
   STEP JogS3:   // S31, max time T#10S, warning time T#7S
              N    #sq.jogDone
   END_STEP
   TRANSITION JogT3 FROM JogS3 TO IndexerHomePos   // T33
      := #signals.releaseNextJog;
   END_TRANSITION
   STEP "Start Grundstellungsfahrt":   // S5, max time T#10S, warning time T#7S
              S    #sq.inHoming
   END_STEP
   TRANSITION GST_Aktiv FROM "Start Grundstellungsfahrt" TO GS_ResetRelease   // T6
      := #ixReleaseHoming AND #signals.releaseCycle;
   END_TRANSITION
   STEP "Fertig Grundstellungsfahrt":   // S6, max time T#10S, warning time T#7S
              R    #sq.inHoming
   END_STEP
   TRANSITION GST_Beendet FROM "Fertig Grundstellungsfahrt" TO Ende   // T7
      := "AlwaysTRUE";
   END_TRANSITION
   STEP Ende:   // S7, max time T#10S, warning time T#7S
          S0  R    #sq.running
   END_STEP
   TRANSITION Beendet FROM Ende TO Grundstellung   // T8, jump
      := "AlwaysTRUE";
   END_TRANSITION
   STEP OpenStopper:   // S17, max time T#10S, warning time T#7S
      supervision V := #OpenStopper.X AND #cylinder_stopper.inError;
              N    #cylinder_stopper.setWorkPos
   END_STEP
   TRANSITION "WT hat Stopper verlassen" FROM OpenStopper TO WaitForTarget   // T18
      := #sinstCarrierLeftIndexer.Q;
   END_TRANSITION
   STEP JogS4:   // S27, max time T#10S, warning time T#7S
              N    #sq.jogDone
   END_STEP
   TRANSITION JogT4 FROM JogS4 TO OpenStopper   // T29
      := #signals.releaseNextJog;
   END_TRANSITION
   STEP OpenGates:   // S30, max time T#10S, warning time T#7S
      supervision V := (#sstReleaseCycle.T >= #itMaxRuntime) OR (("TransportActors".Gate_1.inError OR "TransportActors".Gate_2.inError) AND #OpenGates.X);
              R    "TransportActors".Gate_1.setWorkPos
              R    "TransportActors".Gate_2.setWorkPos
   END_STEP
   TRANSITION GatesOpened FROM OpenGates TO JogS3   // T32
      := "TransportActors".Gate_1.inHomePos AND "TransportActors".Gate_2.inHomePos;
   END_TRANSITION
   STEP Decision:   // S18, max time T#10S, warning time T#7S
   END_STEP
   TRANSITION CarrierIsNotDone FROM Decision TO IndexerWorkPos   // T19
      := NOT #qxCarrierIsDone;
   END_TRANSITION
   TRANSITION CarrierIsDone FROM Decision TO OpenGates   // T20
      := #qxCarrierIsDone;
   END_TRANSITION
   STEP GS_CylHome:   // S14, max time T#10S, warning time T#7S
      supervision V := #GS_CylHome.X AND #cylinder_lift.inError;
              S    #cylinder_lift.setHomePos
              R    #cylinder_lift.setWorkPos
   END_STEP
   TRANSITION "Lift steht in Grundstellung_1" FROM GS_CylHome TO GS_OpenGates   // T15
      := #cylinder_lift.inHomePos;
   END_TRANSITION
   STEP IndexerWorkPos:   // S15, max time T#10S, warning time T#7S
      supervision V := #IndexerWorkPos.X AND #cylinder_lift.inError;
              S    #cylinder_lift.setWorkPos
              R    #cylinder_lift.setHomePos
   END_STEP
   TRANSITION "Lift steht in Arbeitsstellung_1" FROM IndexerWorkPos TO JogS1   // T16
      := #cylinder_lift.inWorkPos;
   END_TRANSITION
   STEP Release:   // S20, max time T#10S, warning time T#7S
          S1  S    #releaseWorkStep
   END_STEP
   TRANSITION WorkstepIsReleased FROM Release TO Ende   // T23
      := true;
   END_TRANSITION
   STEP WaitForTarget:   // S12, max time T#10S, warning time T#7S
      supervision V := #sstReleaseCycle.T >= #itMaxRuntime;
   END_STEP
   TRANSITION TargetIsReached FROM WaitForTarget TO Fertigmeldung   // T13
      := ((#WaitForTarget.U >= t#0s) AND NOT #ixCheckTargetReached) OR #ixTargetReached;
   END_TRANSITION
   STEP JogS1:   // S28, max time T#10S, warning time T#7S
              N    #sq.jogDone
   END_STEP
   TRANSITION JogT1 FROM JogS1 TO CloseGates   // T30
      := #signals.releaseNextJog;
   END_TRANSITION
   STEP CloseGates:   // S29, max time T#10S, warning time T#7S
      supervision V := (#sstReleaseCycle.T >= #itMaxRuntime) OR (("TransportActors".Gate_1.inError OR "TransportActors".Gate_2.inError) AND #CloseGates.X);
              S    "TransportActors".Gate_1.setWorkPos
              S    "TransportActors".Gate_2.setWorkPos
   END_STEP
   TRANSITION GatesClosed FROM CloseGates TO Release   // T31
      := "TransportActors".Gate_1.inWorkPos AND "TransportActors".Gate_2.inWorkPos;
   END_TRANSITION
   STEP Fertigmeldung:   // S4, max time T#10S, warning time T#7S
              S    #sq.done
              R    #qxCarrierIsDone
   END_STEP
   TRANSITION Fertig FROM Fertigmeldung TO Ende   // T4
      := "AlwaysTRUE";
   END_TRANSITION
   STEP IndexerHomePos:   // S16, max time T#10S, warning time T#7S
      supervision V := #IndexerHomePos.X AND #cylinder_lift.inError;
              S    #cylinder_lift.setHomePos
              R    #cylinder_lift.setWorkPos
   END_STEP
   TRANSITION "Lift steht in Arbeitsstellung_2" FROM IndexerHomePos TO JogS4   // T17
      := #cylinder_lift.inHomePos;
   END_TRANSITION
   STEP GS_OpenGates:   // S32, max time T#10S, warning time T#7S
      supervision V := (#sstReleaseCycle.T >= #itMaxRuntime) OR (("TransportActors".Gate_1.inError OR "TransportActors".Gate_2.inError) AND #GS_OpenGates.X);
              R    "TransportActors".Gate_1.setWorkPos
              R    "TransportActors".Gate_2.setWorkPos
   END_STEP
   TRANSITION GS_GatesOpened FROM GS_OpenGates TO "Fertig Grundstellungsfahrt"   // T34
      := "TransportActors".Gate_1.inHomePos AND "TransportActors".Gate_2.inHomePos;
   END_TRANSITION
   STEP GS_ResetRelease:   // S22, max time T#10S, warning time T#7S
              R    #releaseWorkStep
   END_STEP
   TRANSITION GS_ReleaseReseted FROM GS_ResetRelease TO GS_CheckCarrier   // T26
      := NOT #releaseWorkStep;
   END_TRANSITION
   STEP GS_CheckCarrier:   // S23, max time T#10S, warning time T#7S
   END_STEP
   TRANSITION GS_NoCarrier FROM GS_CheckCarrier TO GS_ResetCarrierIsDone   // T27
      := NOT #sinstCarrierOnIndexer.Q;
   END_TRANSITION
   TRANSITION GS_CarrierOnIndexer FROM GS_CheckCarrier TO GS_CylHome   // T28
      := #sinstCarrierOnIndexer.Q;
   END_TRANSITION
   STEP GS_ResetCarrierIsDone:   // S24, max time T#10S, warning time T#7S
              R    #qxCarrierIsDone
   END_STEP
   TRANSITION GS_Reseted FROM GS_ResetCarrierIsDone TO GS_CylHome   // T35
      := true;
   END_TRANSITION

   // permanent post-instructions
   NETWORK 1
   TITLE = Störungssignal weitergeben
      #sq.error := #ERR_FLT;
   NETWORK 2
   TITLE = Ablauf ist aktiv
      #qxIsActive := #sq.running;
   NETWORK 3
   TITLE = steht in Grundstellung
      #qxIsInHome := #sq.inHome AND NOT #sq.running;
   NETWORK 4
   TITLE = WT-Träger ist fertig bearbeitet worden
      #_w1 := NOT #releaseWorkStep AND #sxTrigReleaseWorkStep;   // falling edge
      #sxTrigReleaseWorkStep := #releaseWorkStep;
      IF #_w1 AND NOT #signals.isHoming AND #cylinder_lift.inWorkPos THEN #qxCarrierIsDone := TRUE; END_IF;
END_FUNCTION_BLOCK

FUNCTION "FG10StepSequences" : Void   // FC2010, FBD
TITLE = Schrittkettensteuerung
{ S7_Optimized_Access := 'TRUE' }
VERSION : 0.1
// Ersteller: Andreas Fast Automation
// E-Mail: automation@fast-andreas.de
// 
// Projekt dient zu Demonstrationszwecken und frei genutzt werden.
// 
// Bausteinbeschreibung:
   VAR_IN_OUT
      station : "typeStation";
   END_VAR
   VAR_TEMP
      tempInit : Bool;
      tempAck : Bool;
      tempSwAuto : Bool;
      tempSwMan : Bool;
      tempSwTap : Bool;
      tempPush : Bool;
   END_VAR
BEGIN

REGION Network 1: Graph Parameter
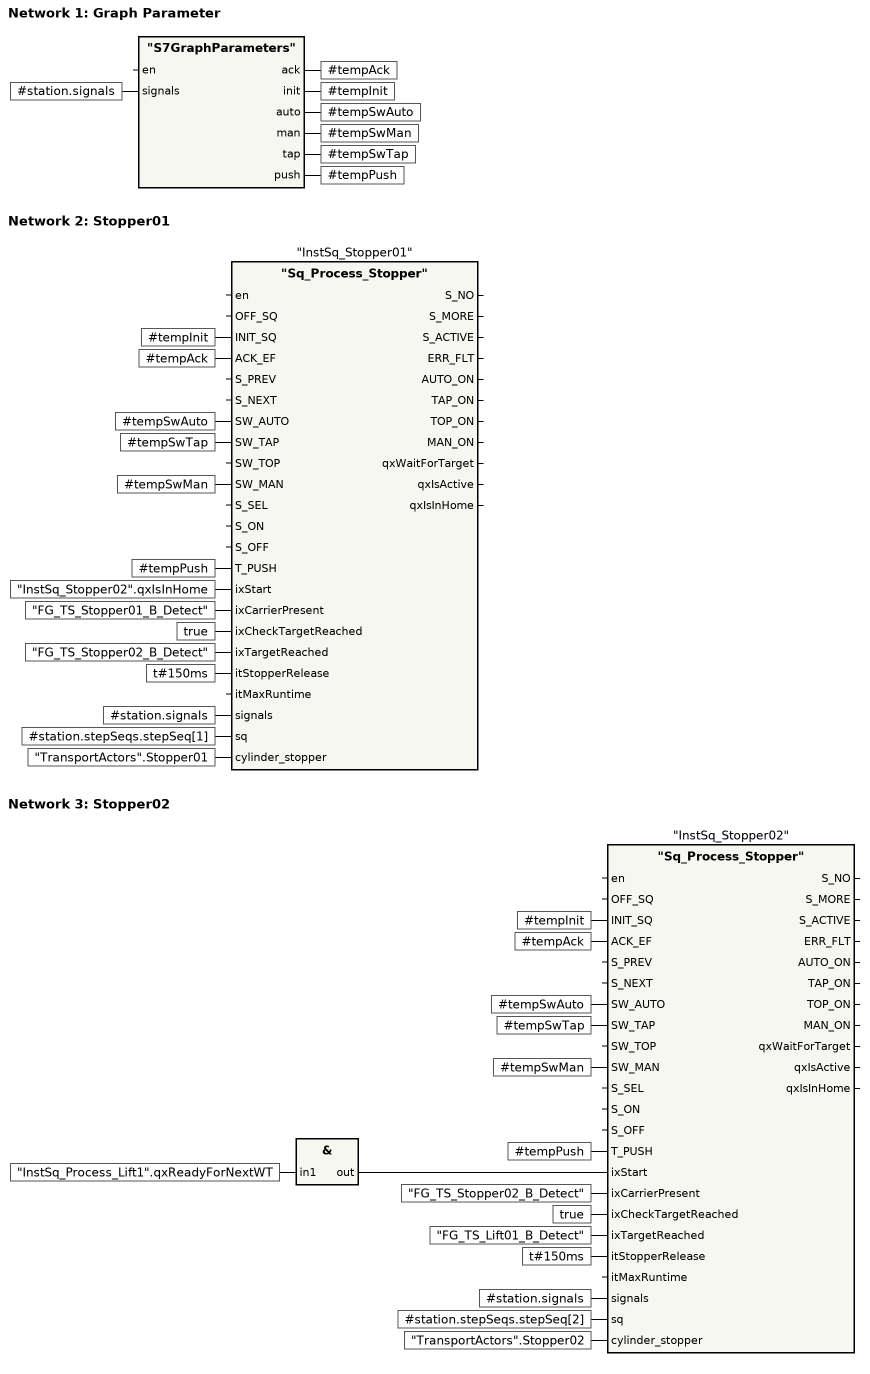
   "S7GraphParameters"(signals := #station.signals,
                       ack => #tempAck,
                       init => #tempInit,
                       auto => #tempSwAuto,
                       man => #tempSwMan,
                       tap => #tempSwTap,
                       push => #tempPush);
END_REGION

REGION Network 2: Stopper01
   "InstSq_Stopper01"(INIT_SQ := #tempInit,   // "Sq_Process_Stopper"
                      ACK_EF := #tempAck,
                      SW_AUTO := #tempSwAuto,
                      SW_TAP := #tempSwTap,
                      SW_MAN := #tempSwMan,
                      T_PUSH := #tempPush,
                      ixStart := "InstSq_Stopper02".qxIsInHome,
                      ixCarrierPresent := "FG_TS_Stopper01_B_Detect",
                      ixCheckTargetReached := true,
                      ixTargetReached := "FG_TS_Stopper02_B_Detect",
                      itStopperRelease := t#150ms,
                      signals := #station.signals,
                      sq := #station.stepSeqs.stepSeq[1],
                      cylinder_stopper := "TransportActors".Stopper01);
END_REGION

